    (*=== VARIABLE LIST ===============================================================================*)
    zz_VariableList :   ARRAY[1..zz_VARIABLECOUNT] OF MBCFG_typVARIABLE :=
    (    DataType        := MBCFG_TYPE_REAL,
        ByteOrder       := MBCFG_BYTE_ORDER_3,
        BitSize         := 32,
        ptVar           := 0,
        ReadJobIndex    := 1,
        ReadStartBitNo  := 256,
        WriteJobIndex   := 0,
        WriteStartBitNo := 0 ),
    (    DataType        := MBCFG_TYPE_REAL,
        ByteOrder       := MBCFG_BYTE_ORDER_3,
        BitSize         := 32,
        ptVar           := 0,
        ReadJobIndex    := 1,
        ReadStartBitNo  := 288,
        WriteJobIndex   := 0,
        WriteStartBitNo := 0 ),
    (    DataType        := MBCFG_TYPE_REAL,
        ByteOrder       := MBCFG_BYTE_ORDER_3,
        BitSize         := 32,
        ptVar           := 0,
        ReadJobIndex    := 1,
        ReadStartBitNo  := 320,
        WriteJobIndex   := 0,
        WriteStartBitNo := 0 ),
    (    DataType        := MBCFG_TYPE_REAL,
        ByteOrder       := MBCFG_BYTE_ORDER_3,
        BitSize         := 32,
        ptVar           := 0,
        ReadJobIndex    := 1,
        ReadStartBitNo  := 384,
        WriteJobIndex   := 0,
        WriteStartBitNo := 0 ),
    (    DataType        := MBCFG_TYPE_REAL,
        ByteOrder       := MBCFG_BYTE_ORDER_3,
        BitSize         := 32,
        ptVar           := 0,
        ReadJobIndex    := 1,
        ReadStartBitNo  := 416,
        WriteJobIndex   := 0,
        WriteStartBitNo := 0 ),
    (    DataType        := MBCFG_TYPE_REAL,
        ByteOrder       := MBCFG_BYTE_ORDER_3,
        BitSize         := 32,
        ptVar           := 0,
        ReadJobIndex    := 1,
        ReadStartBitNo  := 448,
        WriteJobIndex   := 0,
        WriteStartBitNo := 0 ),
    (    DataType        := MBCFG_TYPE_REAL,
        ByteOrder       := MBCFG_BYTE_ORDER_3,
        BitSize         := 32,
        ptVar           := 0,
        ReadJobIndex    := 1,
        ReadStartBitNo  := 0,
        WriteJobIndex   := 0,
        WriteStartBitNo := 0 ),
    (    DataType        := MBCFG_TYPE_REAL,
        ByteOrder       := MBCFG_BYTE_ORDER_3,
        BitSize         := 32,
        ptVar           := 0,
        ReadJobIndex    := 1,
        ReadStartBitNo  := 32,
        WriteJobIndex   := 0,
        WriteStartBitNo := 0 ),
    (    DataType        := MBCFG_TYPE_REAL,
        ByteOrder       := MBCFG_BYTE_ORDER_3,
        BitSize         := 32,
        ptVar           := 0,
        ReadJobIndex    := 1,
        ReadStartBitNo  := 64,
        WriteJobIndex   := 0,
        WriteStartBitNo := 0 ),
    (    DataType        := MBCFG_TYPE_REAL,
        ByteOrder       := MBCFG_BYTE_ORDER_3,
        BitSize         := 32,
        ptVar           := 0,
        ReadJobIndex    := 1,
        ReadStartBitNo  := 96,
        WriteJobIndex   := 0,
        WriteStartBitNo := 0 ),
    (    DataType        := MBCFG_TYPE_REAL,
        ByteOrder       := MBCFG_BYTE_ORDER_3,
        BitSize         := 32,
        ptVar           := 0,
        ReadJobIndex    := 1,
        ReadStartBitNo  := 128,
        WriteJobIndex   := 0,
        WriteStartBitNo := 0 ),
    (    DataType        := MBCFG_TYPE_REAL,
        ByteOrder       := MBCFG_BYTE_ORDER_3,
        BitSize         := 32,
        ptVar           := 0,
        ReadJobIndex    := 1,
        ReadStartBitNo  := 160,
        WriteJobIndex   := 0,
        WriteStartBitNo := 0 ),
    (    DataType        := MBCFG_TYPE_REAL,
        ByteOrder       := MBCFG_BYTE_ORDER_3,
        BitSize         := 32,
        ptVar           := 0,
        ReadJobIndex    := 1,
        ReadStartBitNo  := 192,
        WriteJobIndex   := 0,
        WriteStartBitNo := 0 ),
    (    DataType        := MBCFG_TYPE_REAL,
        ByteOrder       := MBCFG_BYTE_ORDER_3,
        BitSize         := 32,
        ptVar           := 0,
        ReadJobIndex    := 1,
        ReadStartBitNo  := 224,
        WriteJobIndex   := 0,
        WriteStartBitNo := 0 ),
    (    DataType        := MBCFG_TYPE_REAL,
        ByteOrder       := MBCFG_BYTE_ORDER_3,
        BitSize         := 32,
        ptVar           := 0,
        ReadJobIndex    := 2,
        ReadStartBitNo  := 416,
        WriteJobIndex   := 0,
        WriteStartBitNo := 0 ),
    (    DataType        := MBCFG_TYPE_REAL,
        ByteOrder       := MBCFG_BYTE_ORDER_3,
        BitSize         := 32,
        ptVar           := 0,
        ReadJobIndex    := 2,
        ReadStartBitNo  := 0,
        WriteJobIndex   := 0,
        WriteStartBitNo := 0 ),
    (    DataType        := MBCFG_TYPE_REAL,
        ByteOrder       := MBCFG_BYTE_ORDER_3,
        BitSize         := 32,
        ptVar           := 0,
        ReadJobIndex    := 2,
        ReadStartBitNo  := 32,
        WriteJobIndex   := 0,
        WriteStartBitNo := 0 ),
    (    DataType        := MBCFG_TYPE_REAL,
        ByteOrder       := MBCFG_BYTE_ORDER_3,
        BitSize         := 32,
        ptVar           := 0,
        ReadJobIndex    := 2,
        ReadStartBitNo  := 64,
        WriteJobIndex   := 0,
        WriteStartBitNo := 0 ),
    (    DataType        := MBCFG_TYPE_REAL,
        ByteOrder       := MBCFG_BYTE_ORDER_3,
        BitSize         := 32,
        ptVar           := 0,
        ReadJobIndex    := 2,
        ReadStartBitNo  := 256,
        WriteJobIndex   := 0,
        WriteStartBitNo := 0 ),
    (    DataType        := MBCFG_TYPE_REAL,
        ByteOrder       := MBCFG_BYTE_ORDER_3,
        BitSize         := 32,
        ptVar           := 0,
        ReadJobIndex    := 3,
        ReadStartBitNo  := 0,
        WriteJobIndex   := 0,
        WriteStartBitNo := 0 ),
    (    DataType        := MBCFG_TYPE_REAL,
        ByteOrder       := MBCFG_BYTE_ORDER_3,
        BitSize         := 32,
        ptVar           := 0,
        ReadJobIndex    := 3,
        ReadStartBitNo  := 128,
        WriteJobIndex   := 0,
        WriteStartBitNo := 0 )

                        ;
    (*=================================================================================================*)

    (*=== JOB LIST ====================================================================================*)
    zz_JobList     :   ARRAY[1..zz_JOBCOUNT] OF MBCFG_typCOM_JOB :=
     (   Functioncode            := 3,
        ReadStartAddress        := 2053,
        ReadQuantity            := 30,
        WriteStartAddress       := 0,
        WriteQuantity           := 0,
        ptReadData              := 0, 
        ptWriteData             := 0 ),
     (   Functioncode            := 3,
        ReadStartAddress        := 2159,
        ReadQuantity            := 28,
        WriteStartAddress       := 0,
        WriteQuantity           := 0,
        ptReadData              := 0, 
        ptWriteData             := 0 ),
     (   Functioncode            := 3,
        ReadStartAddress        := 2105,
        ReadQuantity            := 10,
        WriteStartAddress       := 0,
        WriteQuantity           := 0,
        ptReadData              := 0, 
        ptWriteData             := 0 )

                        ;
    (*=================================================================================================*)

    (*=== DATA FIELDS =================================================================================*)
     zz_DataField_1_Read       :       ARRAY[1..30] OF WORD;
     zz_DataField_2_Read       :       ARRAY[1..28] OF WORD;
     zz_DataField_3_Read       :       ARRAY[1..10] OF WORD;
	
    (*=================================================================================================*)

    (*=== MODBUS MASTER =====================================*)
    zz_MBCFG_MASTER_ETH :       MBCFG_MASTER_UDP;
    (*=======================================================*)

END_VAR
(*--- for each variable -------------------------*)
   zz_VariableList[1].ptVar := ADR(PactiveL1);
   zz_VariableList[2].ptVar := ADR(PactiveL2);
   zz_VariableList[3].ptVar := ADR(PactiveL3);
   zz_VariableList[4].ptVar := ADR(PreactiveL1);
   zz_VariableList[5].ptVar := ADR(PreactiveL2);
   zz_VariableList[6].ptVar := ADR(PreactiveL3);
   zz_VariableList[7].ptVar := ADR(VoltageL1);
   zz_VariableList[8].ptVar := ADR(VoltageL2);
   zz_VariableList[9].ptVar := ADR(VoltageL3);
   zz_VariableList[10].ptVar := ADR(VoltageL4);
   zz_VariableList[11].ptVar := ADR(PhaseCurrentL1);
   zz_VariableList[12].ptVar := ADR(PhaseCurrentL2);
   zz_VariableList[13].ptVar := ADR(PhaseCurrentL3);
   zz_VariableList[14].ptVar := ADR(PhaseCurrentLN);
   zz_VariableList[15].ptVar := ADR(FieldRotation);
   zz_VariableList[16].ptVar := ADR(CosPihL1);
   zz_VariableList[17].ptVar := ADR(CosPihL2);
   zz_VariableList[18].ptVar := ADR(CosPihL3);
   zz_VariableList[19].ptVar := ADR(Frequency);
   zz_VariableList[20].ptVar := ADR(PactivetTot);
   zz_VariableList[21].ptVar := ADR(PactivetTotL4);

(*-----------------------------------------------*)

(*--- for each job -----------------------------------*)
zz_JobList[1].ptReadData   := ADR(zz_DataField_1_Read);
zz_JobList[2].ptReadData   := ADR(zz_DataField_2_Read);
zz_JobList[3].ptReadData   := ADR(zz_DataField_3_Read);

(*----------------------------------------------------*)


(*#### START OF FIXED CODE #####################################*)
zz_MBCFG_MASTER_ETH(	strIpAddress    := MBCFG_IpAddress,                 (* fixed entry     *)
                        uiPort          := MBCFG_Port,                      (* fixed entry     *)
                        bUnitID         := MBCFG_UnitID,                    (* fixed entry     *)
                        tTimeOut        := MBCFG_TimeOut,                   (* fixed entry     *)
                        iVariableCount  := zz_VARIABLECOUNT,
                        ptVariableList  := ADR(zz_VariableList),
                        iJobCount       := zz_JOBCOUNT,
                        ptJobList       := ADR(zz_JobList),
                        tRequestDelay   := MBCFG_RequestDelay,              (* fixed entry     *)
                        eError          => MBCFG_Error,                     (* fixed entry     *)
                        LastJob         => MBCFG_LastJob                    (* fixed entry     *)
                    );
(*##############################################################*)
END_PROGRAM

(* POU 01. PowerQualityMeasurements/PQ_1, FBD *)
PROGRAM PQ_1
VAR
	abProcessImageInput	AT %IW12			: ARRAY[0..23] OF BYTE;
	abProcessImageOutput 	AT %QW20		: ARRAY[0..23] OF BYTE;

	bToken										: BYTE;

	State_750_495 							: Fb_750_495_State;
		typ_750_495_State 						: typ_750_495_State;

	Configuration_750_495					: Fb_750_495_Configuration;
		typConfig_750_495						: typConfig_750_495;
		xReadyConfig								: BOOL;
		bFeedbackConfig							: BYTE;

	AC_Compact_01_750_495				: Fb_750_495_AC_Compact_01;
		rTotalActivePower							: REAL;
		rTotalReactivePower						: REAL;
		rTotalApparentPower						: REAL;
		rTotalPowerFactorPF						: REAL;
		rTotalActiveEnergy							: REAL;
		rTotalReactiveEnergy						: REAL;
		rTotalApparentEnergy						: REAL;
		rCurrentN									: REAL;
		xRotatingField								: BOOL;
		arCurrent									: ARRAY[1..3] OF REAL;
		axOvercurrent								: ARRAY[1..3] OF BOOL;
		arVoltage_L_N							: ARRAY[1..3] OF REAL;
		axUndervoltage							: ARRAY[1..3] OF BOOL;
		axOvervoltage								: ARRAY[1..3] OF BOOL;
		arActivePower								: ARRAY[1..3] OF REAL;
		arReactivePower							: ARRAY[1..3] OF REAL;
		arApparentPower							: ARRAY[1..3] OF REAL;
		arCosPhi									: ARRAY[1..3] OF REAL;
		arPowerFactorPF							: ARRAY[1..3] OF REAL;
		arFrequency								: ARRAY[1..3] OF REAL;
		axNoZero									: ARRAY[1..3] OF BOOL;
		axVoltSag									: ARRAY[1..3] OF BOOL;
		ai4Quadrant								: ARRAY[1..3] OF INT;

		xReadyCompact_01						: BOOL;
		abFeedbackCompact_01					: ARRAY[1..8] OF BYTE;


END_VAR
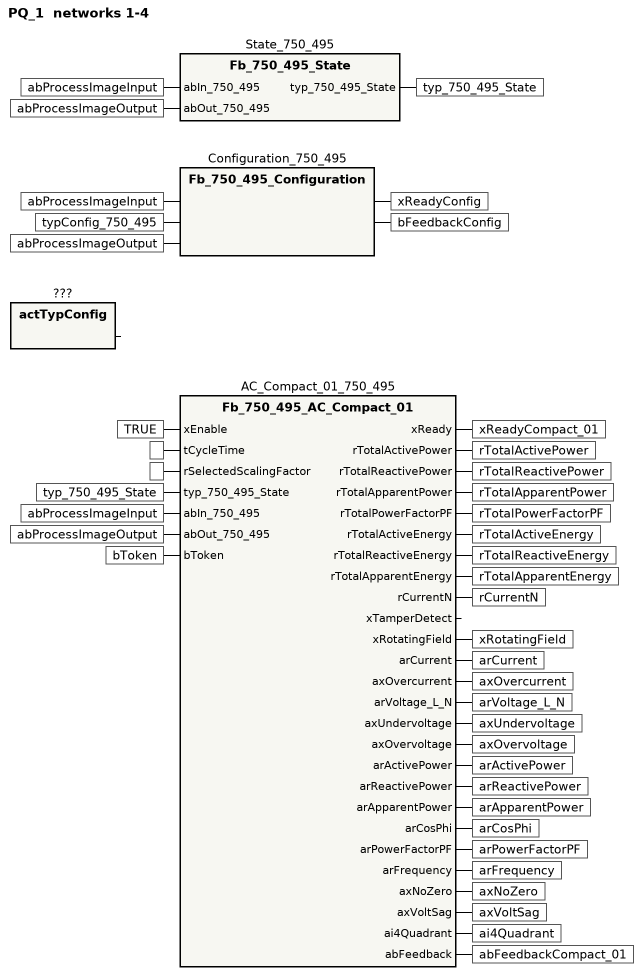
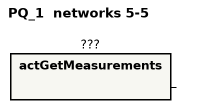
_FBD_ (* Function Block Diagram *)
NETWORK 1
	State_750_495:Fb_750_495_State(abIn_750_495: abProcessImageInput, abOut_750_495: abProcessImageOutput) => typ_750_495_State
NETWORK 2
	Configuration_750_495:Fb_750_495_Configuration(abProcessImageInput, typConfig_750_495, abProcessImageOutput, out 2 => bFeedbackConfig) => xReadyConfig
NETWORK 3
	???:actTypConfig()
NETWORK 4
	AC_Compact_01_750_495:Fb_750_495_AC_Compact_01(xEnable: TRUE, tCycleTime: , rSelectedScalingFactor: , typ_750_495_State: typ_750_495_State, abIn_750_495: abProcessImageInput, abOut_750_495: abProcessImageOutput, bToken: bToken, rTotalActivePower => rTotalActivePower, rTotalReactivePower => rTotalReactivePower, rTotalApparentPower => rTotalApparentPower, rTotalPowerFactorPF => rTotalPowerFactorPF, rTotalActiveEnergy => rTotalActiveEnergy, rTotalReactiveEnergy => rTotalReactiveEnergy, rTotalApparentEnergy => rTotalApparentEnergy, rCurrentN => rCurrentN, xRotatingField => xRotatingField, arCurrent => arCurrent, axOvercurrent => axOvercurrent, arVoltage_L_N => arVoltage_L_N, axUndervoltage => axUndervoltage, axOvervoltage => axOvervoltage, arActivePower => arActivePower, arReactivePower => arReactivePower, arApparentPower => arApparentPower, arCosPhi => arCosPhi, arPowerFactorPF => arPowerFactorPF, arFrequency => arFrequency, axNoZero => axNoZero, axVoltSag => axVoltSag, ai4Quadrant => ai4Quadrant, abFeedback => abFeedbackCompact_01) => xReadyCompact_01
NETWORK 5
	???:actGetMeasurements()
_END_FBD_
(* the same logic as Structured Text *)
(* Network 1 *)
State_750_495(abIn_750_495 := abProcessImageInput, abOut_750_495 := abProcessImageOutput);
typ_750_495_State := State_750_495.typ_750_495_State;
(* Network 2: see the listing above *)
(* Network 3: see the listing above *)
(* Network 4: see the listing above *)
(* Network 5: see the listing above *)
END_PROGRAM
ACTION actGetMeasurements:
arMeasurementsGroup1[1] := arActivePower[1];
arMeasurementsGroup1[2] := arActivePower[2];
arMeasurementsGroup1[3] := arActivePower[3];
arMeasurementsGroup1[4] := arReactivePower[1];
arMeasurementsGroup1[5] := arReactivePower[2];
arMeasurementsGroup1[6] := arReactivePower[3];
arMeasurementsGroup1[7] := arVoltage_L_N[1];
arMeasurementsGroup1[8] := arVoltage_L_N[2];
arMeasurementsGroup1[9] := arVoltage_L_N[3];
arMeasurementsGroup1[10] := arCurrent[1];
arMeasurementsGroup1[11] := arCurrent[2];
arMeasurementsGroup1[12] := arCurrent[3];
arMeasurementsGroup1[13] := arFrequency[1];
arMeasurementsGroup1[14] := arFrequency[2];
arMeasurementsGroup1[15] := arFrequency[3];
arMeasurementsGroup1[16] := rTotalActiveEnergy;
arMeasurementsGroup1[17] := BOOL_TO_REAL(xRotatingField);
arMeasurementsGroup1[18] := rTotalReactiveEnergy;
END_ACTION
ACTION actTypConfig:
typConfig_750_495.typChannelConfig[1].xEnableUserScaling:= TRUE;
typConfig_750_495.typChannelConfig[1].wCurrentTransformerRatio :=CurrentRatioPQ1;

typConfig_750_495.typChannelConfig[2].xEnableUserScaling:= TRUE;
typConfig_750_495.typChannelConfig[2].wCurrentTransformerRatio :=CurrentRatioPQ1;

typConfig_750_495.typChannelConfig[3].xEnableUserScaling:= TRUE;
typConfig_750_495.typChannelConfig[3].wCurrentTransformerRatio :=CurrentRatioPQ1;

typConfig_750_495.xWriteConfig := TRUE;
END_ACTION

(* POU 01. PowerQualityMeasurements/PQ_2, FBD *)
PROGRAM PQ_2
VAR
	abProcessImageInput	AT %IW24			: ARRAY[0..23] OF BYTE;
	abProcessImageOutput 	AT %QW32 			: ARRAY[0..23] OF BYTE;

	bToken										: BYTE;

	State_750_495 							: Fb_750_495_State;
		typ_750_495_State 						: typ_750_495_State;

	Configuration_750_495					: Fb_750_495_Configuration;
		typConfig_750_495						: typConfig_750_495;
		xReadyConfig								: BOOL;
		bFeedbackConfig							: BYTE;

	AC_Compact_01_750_495				: Fb_750_495_AC_Compact_01;
		rTotalActivePower							: REAL;
		rTotalReactivePower						: REAL;
		rTotalApparentPower						: REAL;
		rTotalPowerFactorPF						: REAL;
		rTotalActiveEnergy							: REAL;
		rTotalReactiveEnergy						: REAL;
		rTotalApparentEnergy						: REAL;
		rCurrentN									: REAL;
		xRotatingField								: BOOL;
		arCurrent									: ARRAY[1..3] OF REAL;
		axOvercurrent								: ARRAY[1..3] OF BOOL;
		arVoltage_L_N							: ARRAY[1..3] OF REAL;
		axUndervoltage							: ARRAY[1..3] OF BOOL;
		axOvervoltage								: ARRAY[1..3] OF BOOL;
		arActivePower								: ARRAY[1..3] OF REAL;
		arReactivePower							: ARRAY[1..3] OF REAL;
		arApparentPower							: ARRAY[1..3] OF REAL;
		arCosPhi									: ARRAY[1..3] OF REAL;
		arPowerFactorPF							: ARRAY[1..3] OF REAL;
		arFrequency								: ARRAY[1..3] OF REAL;
		axNoZero									: ARRAY[1..3] OF BOOL;
		axVoltSag									: ARRAY[1..3] OF BOOL;
		ai4Quadrant								: ARRAY[1..3] OF INT;

		xReadyCompact_01						: BOOL;
		abFeedbackCompact_01					: ARRAY[1..8] OF BYTE;


END_VAR
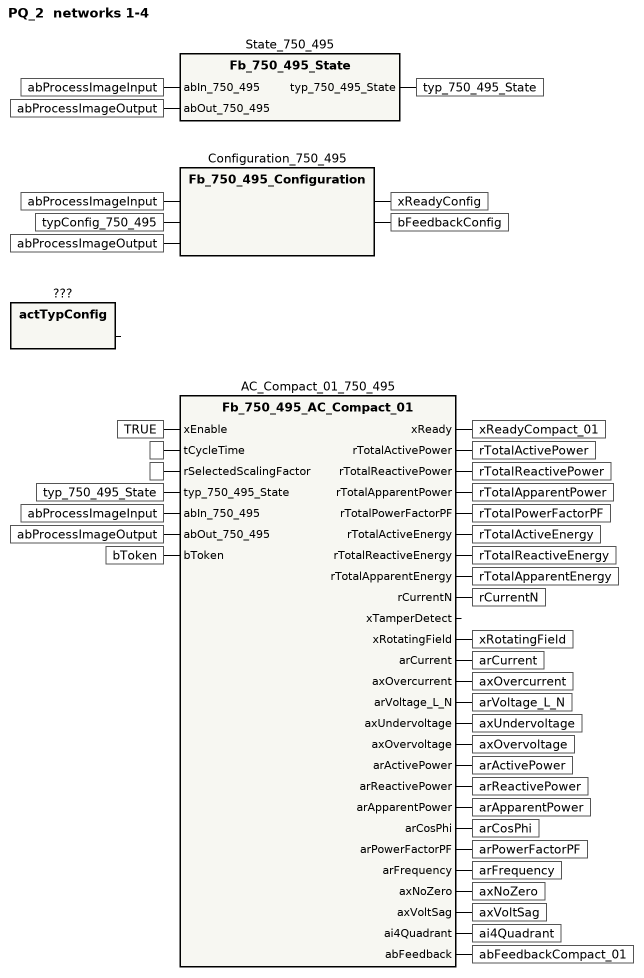
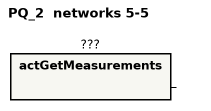
_FBD_ (* Function Block Diagram *)
NETWORK 1
	State_750_495:Fb_750_495_State(abIn_750_495: abProcessImageInput, abOut_750_495: abProcessImageOutput) => typ_750_495_State
NETWORK 2
	Configuration_750_495:Fb_750_495_Configuration(abProcessImageInput, typConfig_750_495, abProcessImageOutput, out 2 => bFeedbackConfig) => xReadyConfig
NETWORK 3
	???:actTypConfig()
NETWORK 4
	AC_Compact_01_750_495:Fb_750_495_AC_Compact_01(xEnable: TRUE, tCycleTime: , rSelectedScalingFactor: , typ_750_495_State: typ_750_495_State, abIn_750_495: abProcessImageInput, abOut_750_495: abProcessImageOutput, bToken: bToken, rTotalActivePower => rTotalActivePower, rTotalReactivePower => rTotalReactivePower, rTotalApparentPower => rTotalApparentPower, rTotalPowerFactorPF => rTotalPowerFactorPF, rTotalActiveEnergy => rTotalActiveEnergy, rTotalReactiveEnergy => rTotalReactiveEnergy, rTotalApparentEnergy => rTotalApparentEnergy, rCurrentN => rCurrentN, xRotatingField => xRotatingField, arCurrent => arCurrent, axOvercurrent => axOvercurrent, arVoltage_L_N => arVoltage_L_N, axUndervoltage => axUndervoltage, axOvervoltage => axOvervoltage, arActivePower => arActivePower, arReactivePower => arReactivePower, arApparentPower => arApparentPower, arCosPhi => arCosPhi, arPowerFactorPF => arPowerFactorPF, arFrequency => arFrequency, axNoZero => axNoZero, axVoltSag => axVoltSag, ai4Quadrant => ai4Quadrant, abFeedback => abFeedbackCompact_01) => xReadyCompact_01
NETWORK 5
	???:actGetMeasurements()
_END_FBD_
(* the same logic as Structured Text *)
(* Network 1 *)
State_750_495(abIn_750_495 := abProcessImageInput, abOut_750_495 := abProcessImageOutput);
typ_750_495_State := State_750_495.typ_750_495_State;
(* Network 2: see the listing above *)
(* Network 3: see the listing above *)
(* Network 4: see the listing above *)
(* Network 5: see the listing above *)
END_PROGRAM
ACTION actGetMeasurements:
arMeasurementsGroup2[1] := arActivePower[1];
arMeasurementsGroup2[2] := arActivePower[2];
arMeasurementsGroup2[3] := arActivePower[3];
arMeasurementsGroup2[4] := arReactivePower[1];
arMeasurementsGroup2[5] := arReactivePower[2];
arMeasurementsGroup2[6] := arReactivePower[3];
arMeasurementsGroup2[7] := arVoltage_L_N[1];
arMeasurementsGroup2[8] := arVoltage_L_N[2];
arMeasurementsGroup2[9] := arVoltage_L_N[3];
arMeasurementsGroup2[10] := arCurrent[1];
arMeasurementsGroup2[11] := arCurrent[2];
arMeasurementsGroup2[12] := arCurrent[3];
arMeasurementsGroup2[13] := arFrequency[1];
arMeasurementsGroup2[14] := arFrequency[2];
arMeasurementsGroup2[15] := arFrequency[3];
arMeasurementsGroup2[16] := rTotalActiveEnergy;
arMeasurementsGroup2[17] := BOOL_TO_REAL(xRotatingField);
arMeasurementsGroup2[18] := rTotalReactiveEnergy;
END_ACTION
ACTION actTypConfig:
typConfig_750_495.typChannelConfig[1].xEnableUserScaling:= TRUE;
typConfig_750_495.typChannelConfig[1].wCurrentTransformerRatio :=CurrentRatioPQ2;

typConfig_750_495.typChannelConfig[2].xEnableUserScaling:= TRUE;
typConfig_750_495.typChannelConfig[2].wCurrentTransformerRatio :=CurrentRatioPQ2;

typConfig_750_495.typChannelConfig[3].xEnableUserScaling:= TRUE;
typConfig_750_495.typChannelConfig[3].wCurrentTransformerRatio :=CurrentRatioPQ2;

typConfig_750_495.xWriteConfig := TRUE;
END_ACTION

(* POU 01. PowerQualityMeasurements/PQ_3, FBD *)
PROGRAM PQ_3
VAR
	abProcessImageInput	AT %IW36			: ARRAY[0..23] OF BYTE;
	abProcessImageOutput 	AT %QW44		: ARRAY[0..23] OF BYTE;

	bToken										: BYTE;

	State_750_495 							: Fb_750_495_State;
		typ_750_495_State 						: typ_750_495_State;

	Configuration_750_495					: Fb_750_495_Configuration;
		typConfig_750_495						: typConfig_750_495;
		xReadyConfig								: BOOL;
		bFeedbackConfig							: BYTE;

	AC_Compact_01_750_495				: Fb_750_495_AC_Compact_01;
		rTotalActivePower							: REAL;
		rTotalReactivePower						: REAL;
		rTotalApparentPower						: REAL;
		rTotalPowerFactorPF						: REAL;
		rTotalActiveEnergy							: REAL;
		rTotalReactiveEnergy						: REAL;
		rTotalApparentEnergy						: REAL;
		rCurrentN									: REAL;
		xRotatingField								: BOOL;
		arCurrent									: ARRAY[1..3] OF REAL;
		axOvercurrent								: ARRAY[1..3] OF BOOL;
		arVoltage_L_N							: ARRAY[1..3] OF REAL;
		axUndervoltage							: ARRAY[1..3] OF BOOL;
		axOvervoltage								: ARRAY[1..3] OF BOOL;
		arActivePower								: ARRAY[1..3] OF REAL;
		arReactivePower							: ARRAY[1..3] OF REAL;
		arApparentPower							: ARRAY[1..3] OF REAL;
		arCosPhi									: ARRAY[1..3] OF REAL;
		arPowerFactorPF							: ARRAY[1..3] OF REAL;
		arFrequency								: ARRAY[1..3] OF REAL;
		axNoZero									: ARRAY[1..3] OF BOOL;
		axVoltSag									: ARRAY[1..3] OF BOOL;
		ai4Quadrant								: ARRAY[1..3] OF INT;

		xReadyCompact_01						: BOOL;
		abFeedbackCompact_01					: ARRAY[1..8] OF BYTE;


END_VAR
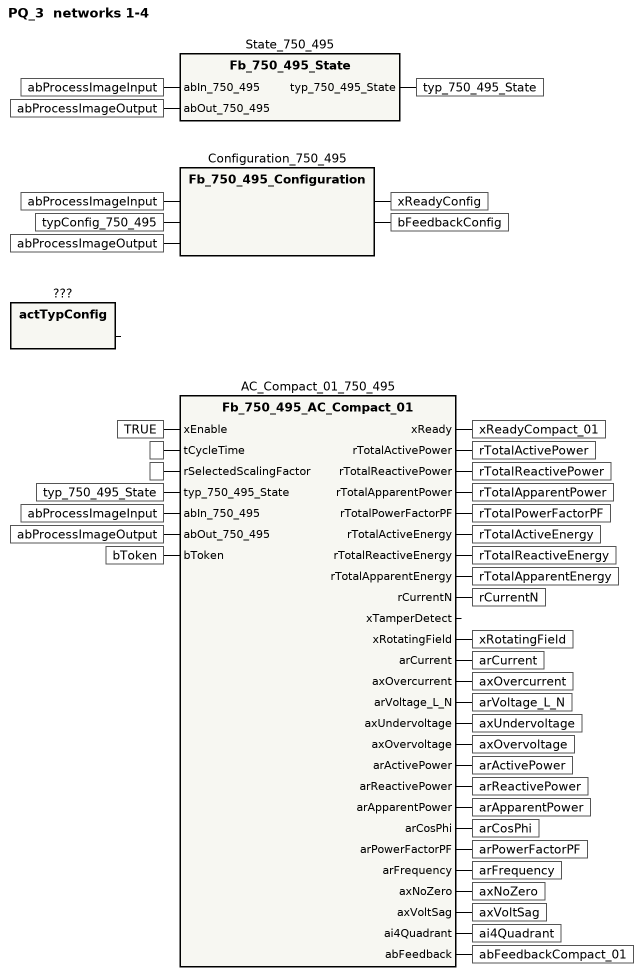
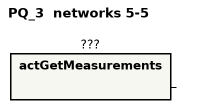
_FBD_ (* Function Block Diagram *)
NETWORK 1
	State_750_495:Fb_750_495_State(abIn_750_495: abProcessImageInput, abOut_750_495: abProcessImageOutput) => typ_750_495_State
NETWORK 2
	Configuration_750_495:Fb_750_495_Configuration(abProcessImageInput, typConfig_750_495, abProcessImageOutput, out 2 => bFeedbackConfig) => xReadyConfig
NETWORK 3
	???:actTypConfig()
NETWORK 4
	AC_Compact_01_750_495:Fb_750_495_AC_Compact_01(xEnable: TRUE, tCycleTime: , rSelectedScalingFactor: , typ_750_495_State: typ_750_495_State, abIn_750_495: abProcessImageInput, abOut_750_495: abProcessImageOutput, bToken: bToken, rTotalActivePower => rTotalActivePower, rTotalReactivePower => rTotalReactivePower, rTotalApparentPower => rTotalApparentPower, rTotalPowerFactorPF => rTotalPowerFactorPF, rTotalActiveEnergy => rTotalActiveEnergy, rTotalReactiveEnergy => rTotalReactiveEnergy, rTotalApparentEnergy => rTotalApparentEnergy, rCurrentN => rCurrentN, xRotatingField => xRotatingField, arCurrent => arCurrent, axOvercurrent => axOvercurrent, arVoltage_L_N => arVoltage_L_N, axUndervoltage => axUndervoltage, axOvervoltage => axOvervoltage, arActivePower => arActivePower, arReactivePower => arReactivePower, arApparentPower => arApparentPower, arCosPhi => arCosPhi, arPowerFactorPF => arPowerFactorPF, arFrequency => arFrequency, axNoZero => axNoZero, axVoltSag => axVoltSag, ai4Quadrant => ai4Quadrant, abFeedback => abFeedbackCompact_01) => xReadyCompact_01
NETWORK 5
	???:actGetMeasurements()
_END_FBD_
(* the same logic as Structured Text *)
(* Network 1 *)
State_750_495(abIn_750_495 := abProcessImageInput, abOut_750_495 := abProcessImageOutput);
typ_750_495_State := State_750_495.typ_750_495_State;
(* Network 2: see the listing above *)
(* Network 3: see the listing above *)
(* Network 4: see the listing above *)
(* Network 5: see the listing above *)
END_PROGRAM
ACTION actGetMeasurements:
arMeasurementsGroup3[1] := arActivePower[1];
arMeasurementsGroup3[2] := arActivePower[2];
arMeasurementsGroup3[3] := arActivePower[3];
arMeasurementsGroup3[4] := arReactivePower[1];
arMeasurementsGroup3[5] := arReactivePower[2];
arMeasurementsGroup3[6] := arReactivePower[3];
arMeasurementsGroup3[7] := arVoltage_L_N[1];
arMeasurementsGroup3[8] := arVoltage_L_N[2];
arMeasurementsGroup3[9] := arVoltage_L_N[3];
arMeasurementsGroup3[10] := arCurrent[1];
arMeasurementsGroup3[11] := arCurrent[2];
arMeasurementsGroup3[12] := arCurrent[3];
arMeasurementsGroup3[13] := arFrequency[1];
arMeasurementsGroup3[14] := arFrequency[2];
arMeasurementsGroup3[15] := arFrequency[3];
arMeasurementsGroup3[16] := rTotalActiveEnergy;
arMeasurementsGroup3[17] := BOOL_TO_REAL(xRotatingField);
arMeasurementsGroup3[18] := rTotalReactiveEnergy;
END_ACTION
ACTION actTypConfig:
typConfig_750_495.typChannelConfig[1].xEnableUserScaling:= TRUE;
typConfig_750_495.typChannelConfig[1].wCurrentTransformerRatio :=CurrentRatioPQ3;

typConfig_750_495.typChannelConfig[2].xEnableUserScaling:= TRUE;
typConfig_750_495.typChannelConfig[2].wCurrentTransformerRatio :=CurrentRatioPQ3;

typConfig_750_495.typChannelConfig[3].xEnableUserScaling:= TRUE;
typConfig_750_495.typChannelConfig[3].wCurrentTransformerRatio :=CurrentRatioPQ3;

typConfig_750_495.xWriteConfig := TRUE;
END_ACTION

(* POU 01. PowerQualityMeasurements/PQ_4, FBD *)
PROGRAM PQ_4
VAR
	abProcessImageInput	AT %IW48			: ARRAY[0..23] OF BYTE;
	abProcessImageOutput 	AT %QW56		: ARRAY[0..23] OF BYTE;

	bToken										: BYTE;

	State_750_495 							: Fb_750_495_State;
		typ_750_495_State 						: typ_750_495_State;

	Configuration_750_495					: Fb_750_495_Configuration;
		typConfig_750_495						: typConfig_750_495;
		xReadyConfig								: BOOL;
		bFeedbackConfig							: BYTE;

	AC_Compact_01_750_495				: Fb_750_495_AC_Compact_01;
		rTotalActivePower							: REAL;
		rTotalReactivePower						: REAL;
		rTotalApparentPower						: REAL;
		rTotalPowerFactorPF						: REAL;
		rTotalActiveEnergy							: REAL;
		rTotalReactiveEnergy						: REAL;
		rTotalApparentEnergy						: REAL;
		rCurrentN									: REAL;
		xRotatingField								: BOOL;
		arCurrent									: ARRAY[1..3] OF REAL;
		axOvercurrent								: ARRAY[1..3] OF BOOL;
		arVoltage_L_N							: ARRAY[1..3] OF REAL;
		axUndervoltage							: ARRAY[1..3] OF BOOL;
		axOvervoltage								: ARRAY[1..3] OF BOOL;
		arActivePower								: ARRAY[1..3] OF REAL;
		arReactivePower							: ARRAY[1..3] OF REAL;
		arApparentPower							: ARRAY[1..3] OF REAL;
		arCosPhi									: ARRAY[1..3] OF REAL;
		arPowerFactorPF							: ARRAY[1..3] OF REAL;
		arFrequency								: ARRAY[1..3] OF REAL;
		axNoZero									: ARRAY[1..3] OF BOOL;
		axVoltSag									: ARRAY[1..3] OF BOOL;
		ai4Quadrant								: ARRAY[1..3] OF INT;

		xReadyCompact_01						: BOOL;
		abFeedbackCompact_01					: ARRAY[1..8] OF BYTE;


END_VAR
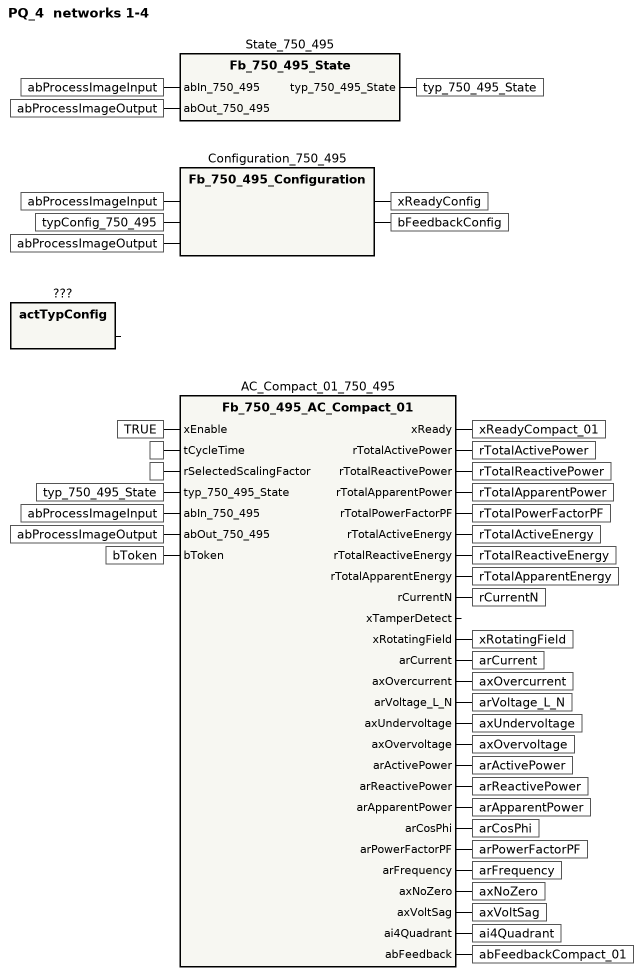
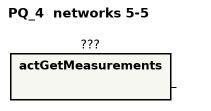
_FBD_ (* Function Block Diagram *)
NETWORK 1
	State_750_495:Fb_750_495_State(abIn_750_495: abProcessImageInput, abOut_750_495: abProcessImageOutput) => typ_750_495_State
NETWORK 2
	Configuration_750_495:Fb_750_495_Configuration(abProcessImageInput, typConfig_750_495, abProcessImageOutput, out 2 => bFeedbackConfig) => xReadyConfig
NETWORK 3
	???:actTypConfig()
NETWORK 4
	AC_Compact_01_750_495:Fb_750_495_AC_Compact_01(xEnable: TRUE, tCycleTime: , rSelectedScalingFactor: , typ_750_495_State: typ_750_495_State, abIn_750_495: abProcessImageInput, abOut_750_495: abProcessImageOutput, bToken: bToken, rTotalActivePower => rTotalActivePower, rTotalReactivePower => rTotalReactivePower, rTotalApparentPower => rTotalApparentPower, rTotalPowerFactorPF => rTotalPowerFactorPF, rTotalActiveEnergy => rTotalActiveEnergy, rTotalReactiveEnergy => rTotalReactiveEnergy, rTotalApparentEnergy => rTotalApparentEnergy, rCurrentN => rCurrentN, xRotatingField => xRotatingField, arCurrent => arCurrent, axOvercurrent => axOvercurrent, arVoltage_L_N => arVoltage_L_N, axUndervoltage => axUndervoltage, axOvervoltage => axOvervoltage, arActivePower => arActivePower, arReactivePower => arReactivePower, arApparentPower => arApparentPower, arCosPhi => arCosPhi, arPowerFactorPF => arPowerFactorPF, arFrequency => arFrequency, axNoZero => axNoZero, axVoltSag => axVoltSag, ai4Quadrant => ai4Quadrant, abFeedback => abFeedbackCompact_01) => xReadyCompact_01
NETWORK 5
	???:actGetMeasurements()
_END_FBD_
(* the same logic as Structured Text *)
(* Network 1 *)
State_750_495(abIn_750_495 := abProcessImageInput, abOut_750_495 := abProcessImageOutput);
typ_750_495_State := State_750_495.typ_750_495_State;
(* Network 2: see the listing above *)
(* Network 3: see the listing above *)
(* Network 4: see the listing above *)
(* Network 5: see the listing above *)
END_PROGRAM
ACTION actGetMeasurements:
arMeasurementsGroup4[1] := arActivePower[1];
arMeasurementsGroup4[2] := arActivePower[2];
arMeasurementsGroup4[3] := arActivePower[3];
arMeasurementsGroup4[4] := arReactivePower[1];
arMeasurementsGroup4[5] := arReactivePower[2];
arMeasurementsGroup4[6] := arReactivePower[3];
arMeasurementsGroup4[7] := arVoltage_L_N[1];
arMeasurementsGroup4[8] := arVoltage_L_N[2];
arMeasurementsGroup4[9] := arVoltage_L_N[3];
arMeasurementsGroup4[10] := arCurrent[1];
arMeasurementsGroup4[11] := arCurrent[2];
arMeasurementsGroup4[12] := arCurrent[3];
arMeasurementsGroup4[13] := arFrequency[1];
arMeasurementsGroup4[14] := arFrequency[2];
arMeasurementsGroup4[15] := arFrequency[3];
arMeasurementsGroup4[16] := rTotalActiveEnergy;
arMeasurementsGroup4[17] := BOOL_TO_REAL(xRotatingField);
arMeasurementsGroup4[18] := rTotalReactiveEnergy;
END_ACTION
ACTION actTypConfig:
typConfig_750_495.typChannelConfig[1].xEnableUserScaling:= TRUE;
typConfig_750_495.typChannelConfig[1].wCurrentTransformerRatio :=CurrentRatioPQ4;

typConfig_750_495.typChannelConfig[2].xEnableUserScaling:= TRUE;
typConfig_750_495.typChannelConfig[2].wCurrentTransformerRatio :=CurrentRatioPQ4;

typConfig_750_495.typChannelConfig[3].xEnableUserScaling:= TRUE;
typConfig_750_495.typChannelConfig[3].wCurrentTransformerRatio :=CurrentRatioPQ4;

typConfig_750_495.xWriteConfig := TRUE;
END_ACTION

(* POU 01. PowerQualityMeasurements/PQ_5, FBD *)
PROGRAM PQ_5
VAR
	abProcessImageInput	AT %IW60			: ARRAY[0..23] OF BYTE;
	abProcessImageOutput 	AT %QW68		: ARRAY[0..23] OF BYTE;

	bToken										: BYTE;

	State_750_495 							: Fb_750_495_State;
		typ_750_495_State 						: typ_750_495_State;

	Configuration_750_495					: Fb_750_495_Configuration;
		typConfig_750_495						: typConfig_750_495;
		xReadyConfig								: BOOL;
		bFeedbackConfig							: BYTE;

	AC_Compact_01_750_495				: Fb_750_495_AC_Compact_01;
		rTotalActivePower							: REAL;
		rTotalReactivePower						: REAL;
		rTotalApparentPower						: REAL;
		rTotalPowerFactorPF						: REAL;
		rTotalActiveEnergy							: REAL;
		rTotalReactiveEnergy						: REAL;
		rTotalApparentEnergy						: REAL;
		rCurrentN									: REAL;
		xRotatingField								: BOOL;
		arCurrent									: ARRAY[1..3] OF REAL;
		axOvercurrent								: ARRAY[1..3] OF BOOL;
		arVoltage_L_N							: ARRAY[1..3] OF REAL;
		axUndervoltage							: ARRAY[1..3] OF BOOL;
		axOvervoltage								: ARRAY[1..3] OF BOOL;
		arActivePower								: ARRAY[1..3] OF REAL;
		arReactivePower							: ARRAY[1..3] OF REAL;
		arApparentPower							: ARRAY[1..3] OF REAL;
		arCosPhi									: ARRAY[1..3] OF REAL;
		arPowerFactorPF							: ARRAY[1..3] OF REAL;
		arFrequency								: ARRAY[1..3] OF REAL;
		axNoZero									: ARRAY[1..3] OF BOOL;
		axVoltSag									: ARRAY[1..3] OF BOOL;
		ai4Quadrant								: ARRAY[1..3] OF INT;

		xReadyCompact_01						: BOOL;
		abFeedbackCompact_01					: ARRAY[1..8] OF BYTE;


END_VAR
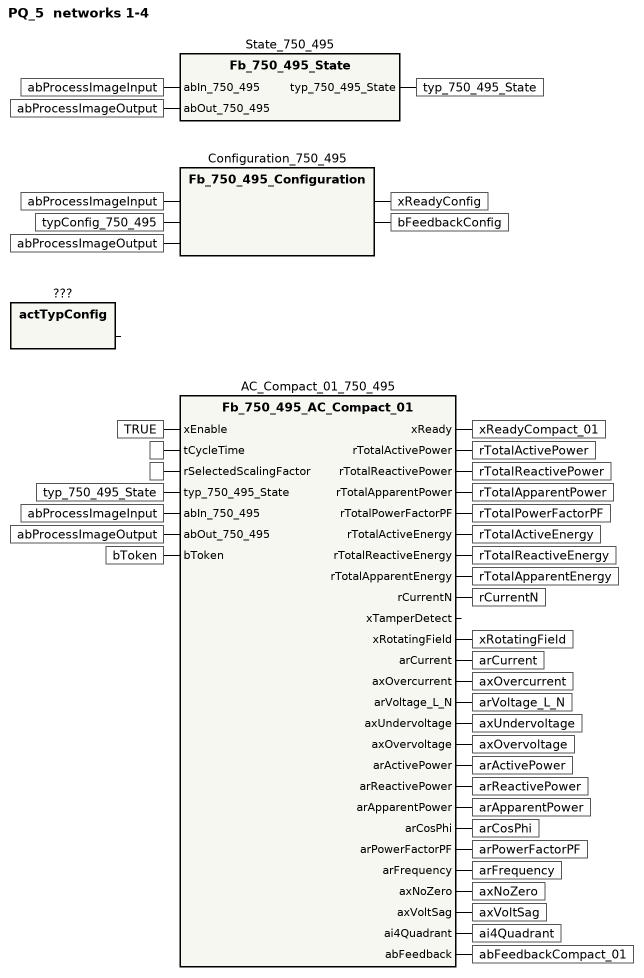
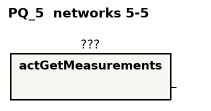
_FBD_ (* Function Block Diagram *)
NETWORK 1
	State_750_495:Fb_750_495_State(abIn_750_495: abProcessImageInput, abOut_750_495: abProcessImageOutput) => typ_750_495_State
NETWORK 2
	Configuration_750_495:Fb_750_495_Configuration(abProcessImageInput, typConfig_750_495, abProcessImageOutput, out 2 => bFeedbackConfig) => xReadyConfig
NETWORK 3
	???:actTypConfig()
NETWORK 4
	AC_Compact_01_750_495:Fb_750_495_AC_Compact_01(xEnable: TRUE, tCycleTime: , rSelectedScalingFactor: , typ_750_495_State: typ_750_495_State, abIn_750_495: abProcessImageInput, abOut_750_495: abProcessImageOutput, bToken: bToken, rTotalActivePower => rTotalActivePower, rTotalReactivePower => rTotalReactivePower, rTotalApparentPower => rTotalApparentPower, rTotalPowerFactorPF => rTotalPowerFactorPF, rTotalActiveEnergy => rTotalActiveEnergy, rTotalReactiveEnergy => rTotalReactiveEnergy, rTotalApparentEnergy => rTotalApparentEnergy, rCurrentN => rCurrentN, xRotatingField => xRotatingField, arCurrent => arCurrent, axOvercurrent => axOvercurrent, arVoltage_L_N => arVoltage_L_N, axUndervoltage => axUndervoltage, axOvervoltage => axOvervoltage, arActivePower => arActivePower, arReactivePower => arReactivePower, arApparentPower => arApparentPower, arCosPhi => arCosPhi, arPowerFactorPF => arPowerFactorPF, arFrequency => arFrequency, axNoZero => axNoZero, axVoltSag => axVoltSag, ai4Quadrant => ai4Quadrant, abFeedback => abFeedbackCompact_01) => xReadyCompact_01
NETWORK 5
	???:actGetMeasurements()
_END_FBD_
(* the same logic as Structured Text *)
(* Network 1 *)
State_750_495(abIn_750_495 := abProcessImageInput, abOut_750_495 := abProcessImageOutput);
typ_750_495_State := State_750_495.typ_750_495_State;
(* Network 2: see the listing above *)
(* Network 3: see the listing above *)
(* Network 4: see the listing above *)
(* Network 5: see the listing above *)
END_PROGRAM
ACTION actGetMeasurements:
arMeasurementsGroup5[1] := arActivePower[1];
arMeasurementsGroup5[2] := arActivePower[2];
arMeasurementsGroup5[3] := arActivePower[3];
arMeasurementsGroup5[4] := arReactivePower[1];
arMeasurementsGroup5[5] := arReactivePower[2];
arMeasurementsGroup5[6] := arReactivePower[3];
arMeasurementsGroup5[7] := arVoltage_L_N[1];
arMeasurementsGroup5[8] := arVoltage_L_N[2];
arMeasurementsGroup5[9] := arVoltage_L_N[3];
arMeasurementsGroup5[10] := arCurrent[1];
arMeasurementsGroup5[11] := arCurrent[2];
arMeasurementsGroup5[12] := arCurrent[3];
arMeasurementsGroup5[13] := arFrequency[1];
arMeasurementsGroup5[14] := arFrequency[2];
arMeasurementsGroup5[15] := arFrequency[3];
arMeasurementsGroup5[16] := rTotalActiveEnergy;
arMeasurementsGroup5[17] := BOOL_TO_REAL(xRotatingField);
arMeasurementsGroup5[18] := rTotalReactiveEnergy;
END_ACTION
ACTION actTypConfig:
typConfig_750_495.typChannelConfig[1].xEnableUserScaling:= TRUE;
typConfig_750_495.typChannelConfig[1].wCurrentTransformerRatio :=CurrentRatioPQ5;

typConfig_750_495.typChannelConfig[2].xEnableUserScaling:= TRUE;
typConfig_750_495.typChannelConfig[2].wCurrentTransformerRatio :=CurrentRatioPQ5;

typConfig_750_495.typChannelConfig[3].xEnableUserScaling:= TRUE;
typConfig_750_495.typChannelConfig[3].wCurrentTransformerRatio :=CurrentRatioPQ5;

typConfig_750_495.xWriteConfig := TRUE;
END_ACTION

(* POU 01. PowerQualityMeasurements/PQ_6, FBD *)
PROGRAM PQ_6
VAR
	abProcessImageInput	AT %IW72			: ARRAY[0..23] OF BYTE;
	abProcessImageOutput 	AT %QW80		: ARRAY[0..23] OF BYTE;

	bToken										: BYTE;

	State_750_495 							: Fb_750_495_State;
		typ_750_495_State 						: typ_750_495_State;

	Configuration_750_495					: Fb_750_495_Configuration;
		typConfig_750_495						: typConfig_750_495;
		xReadyConfig								: BOOL;
		bFeedbackConfig							: BYTE;

	AC_Compact_01_750_495				: Fb_750_495_AC_Compact_01;
		rTotalActivePower							: REAL;
		rTotalReactivePower						: REAL;
		rTotalApparentPower						: REAL;
		rTotalPowerFactorPF						: REAL;
		rTotalActiveEnergy							: REAL;
		rTotalReactiveEnergy						: REAL;
		rTotalApparentEnergy						: REAL;
		rCurrentN									: REAL;
		xRotatingField								: BOOL;
		arCurrent									: ARRAY[1..3] OF REAL;
		axOvercurrent								: ARRAY[1..3] OF BOOL;
		arVoltage_L_N							: ARRAY[1..3] OF REAL;
		axUndervoltage							: ARRAY[1..3] OF BOOL;
		axOvervoltage								: ARRAY[1..3] OF BOOL;
		arActivePower								: ARRAY[1..3] OF REAL;
		arReactivePower							: ARRAY[1..3] OF REAL;
		arApparentPower							: ARRAY[1..3] OF REAL;
		arCosPhi									: ARRAY[1..3] OF REAL;
		arPowerFactorPF							: ARRAY[1..3] OF REAL;
		arFrequency								: ARRAY[1..3] OF REAL;
		axNoZero									: ARRAY[1..3] OF BOOL;
		axVoltSag									: ARRAY[1..3] OF BOOL;
		ai4Quadrant								: ARRAY[1..3] OF INT;

		xReadyCompact_01						: BOOL;
		abFeedbackCompact_01					: ARRAY[1..8] OF BYTE;


END_VAR
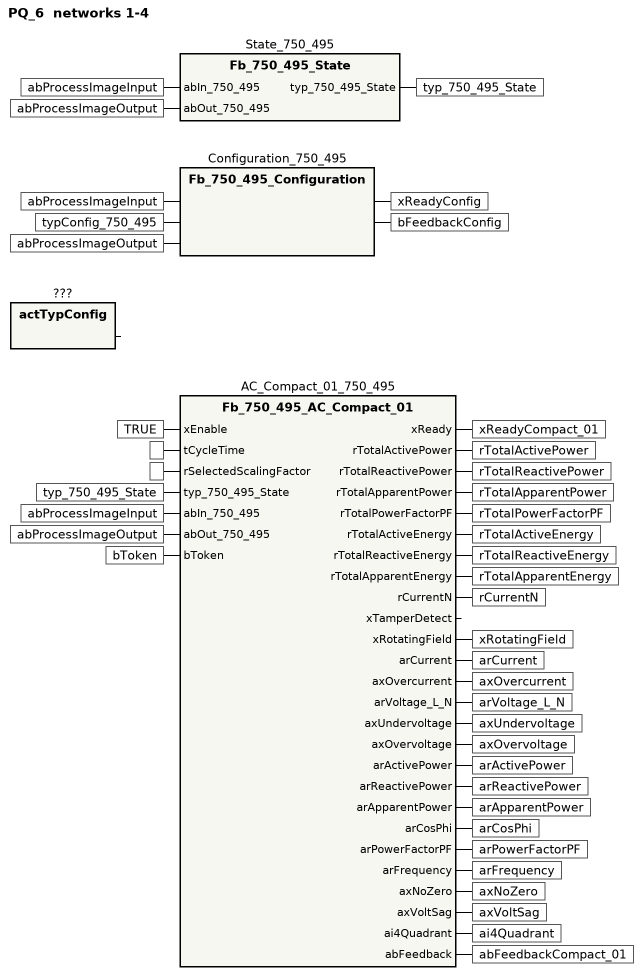
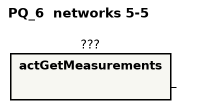
_FBD_ (* Function Block Diagram *)
NETWORK 1
	State_750_495:Fb_750_495_State(abIn_750_495: abProcessImageInput, abOut_750_495: abProcessImageOutput) => typ_750_495_State
NETWORK 2
	Configuration_750_495:Fb_750_495_Configuration(abProcessImageInput, typConfig_750_495, abProcessImageOutput, out 2 => bFeedbackConfig) => xReadyConfig
NETWORK 3
	???:actTypConfig()
NETWORK 4
	AC_Compact_01_750_495:Fb_750_495_AC_Compact_01(xEnable: TRUE, tCycleTime: , rSelectedScalingFactor: , typ_750_495_State: typ_750_495_State, abIn_750_495: abProcessImageInput, abOut_750_495: abProcessImageOutput, bToken: bToken, rTotalActivePower => rTotalActivePower, rTotalReactivePower => rTotalReactivePower, rTotalApparentPower => rTotalApparentPower, rTotalPowerFactorPF => rTotalPowerFactorPF, rTotalActiveEnergy => rTotalActiveEnergy, rTotalReactiveEnergy => rTotalReactiveEnergy, rTotalApparentEnergy => rTotalApparentEnergy, rCurrentN => rCurrentN, xRotatingField => xRotatingField, arCurrent => arCurrent, axOvercurrent => axOvercurrent, arVoltage_L_N => arVoltage_L_N, axUndervoltage => axUndervoltage, axOvervoltage => axOvervoltage, arActivePower => arActivePower, arReactivePower => arReactivePower, arApparentPower => arApparentPower, arCosPhi => arCosPhi, arPowerFactorPF => arPowerFactorPF, arFrequency => arFrequency, axNoZero => axNoZero, axVoltSag => axVoltSag, ai4Quadrant => ai4Quadrant, abFeedback => abFeedbackCompact_01) => xReadyCompact_01
NETWORK 5
	???:actGetMeasurements()
_END_FBD_
(* the same logic as Structured Text *)
(* Network 1 *)
State_750_495(abIn_750_495 := abProcessImageInput, abOut_750_495 := abProcessImageOutput);
typ_750_495_State := State_750_495.typ_750_495_State;
(* Network 2: see the listing above *)
(* Network 3: see the listing above *)
(* Network 4: see the listing above *)
(* Network 5: see the listing above *)
END_PROGRAM
ACTION actGetMeasurements:
arMeasurementsGroup6[1] := arActivePower[1];
arMeasurementsGroup6[2] := arActivePower[2];
arMeasurementsGroup6[3] := arActivePower[3];
arMeasurementsGroup6[4] := arReactivePower[1];
arMeasurementsGroup6[5] := arReactivePower[2];
arMeasurementsGroup6[6] := arReactivePower[3];
arMeasurementsGroup6[7] := arVoltage_L_N[1];
arMeasurementsGroup6[8] := arVoltage_L_N[2];
arMeasurementsGroup6[9] := arVoltage_L_N[3];
arMeasurementsGroup6[10] := arCurrent[1];
arMeasurementsGroup6[11] := arCurrent[2];
arMeasurementsGroup6[12] := arCurrent[3];
arMeasurementsGroup6[13] := arFrequency[1];
arMeasurementsGroup6[14] := arFrequency[2];
arMeasurementsGroup6[15] := arFrequency[3];
arMeasurementsGroup6[16] := rTotalActiveEnergy;
arMeasurementsGroup6[17] := BOOL_TO_REAL(xRotatingField);
arMeasurementsGroup6[18] := rTotalReactiveEnergy;
END_ACTION
ACTION actTypConfig:
typConfig_750_495.typChannelConfig[1].xEnableUserScaling:= TRUE;
typConfig_750_495.typChannelConfig[1].wCurrentTransformerRatio :=CurrentRatioPQ6;

typConfig_750_495.typChannelConfig[2].xEnableUserScaling:= TRUE;
typConfig_750_495.typChannelConfig[2].wCurrentTransformerRatio :=CurrentRatioPQ6;

typConfig_750_495.typChannelConfig[3].xEnableUserScaling:= TRUE;
typConfig_750_495.typChannelConfig[3].wCurrentTransformerRatio :=CurrentRatioPQ6;

typConfig_750_495.xWriteConfig := TRUE;
END_ACTION

(* POU 01. PowerQualityMeasurements/PQ_7, FBD *)
PROGRAM PQ_7
VAR
	abProcessImageInput	AT %IW84			: ARRAY[0..23] OF BYTE;
	abProcessImageOutput 	AT %QW92 			: ARRAY[0..23] OF BYTE;

	bToken										: BYTE;

	State_750_495 							: Fb_750_495_State;
		typ_750_495_State 						: typ_750_495_State;

	Configuration_750_495					: Fb_750_495_Configuration;
		typConfig_750_495						: typConfig_750_495;
		xReadyConfig								: BOOL;
		bFeedbackConfig							: BYTE;

	AC_Compact_01_750_495				: Fb_750_495_AC_Compact_01;
		rTotalActivePower							: REAL;
		rTotalReactivePower						: REAL;
		rTotalApparentPower						: REAL;
		rTotalPowerFactorPF						: REAL;
		rTotalActiveEnergy							: REAL;
		rTotalReactiveEnergy						: REAL;
		rTotalApparentEnergy						: REAL;
		rCurrentN									: REAL;
		xRotatingField								: BOOL;
		arCurrent									: ARRAY[1..3] OF REAL;
		axOvercurrent								: ARRAY[1..3] OF BOOL;
		arVoltage_L_N							: ARRAY[1..3] OF REAL;
		axUndervoltage							: ARRAY[1..3] OF BOOL;
		axOvervoltage								: ARRAY[1..3] OF BOOL;
		arActivePower								: ARRAY[1..3] OF REAL;
		arReactivePower							: ARRAY[1..3] OF REAL;
		arApparentPower							: ARRAY[1..3] OF REAL;
		arCosPhi									: ARRAY[1..3] OF REAL;
		arPowerFactorPF							: ARRAY[1..3] OF REAL;
		arFrequency								: ARRAY[1..3] OF REAL;
		axNoZero									: ARRAY[1..3] OF BOOL;
		axVoltSag									: ARRAY[1..3] OF BOOL;
		ai4Quadrant								: ARRAY[1..3] OF INT;

		xReadyCompact_01						: BOOL;
		abFeedbackCompact_01					: ARRAY[1..8] OF BYTE;


END_VAR
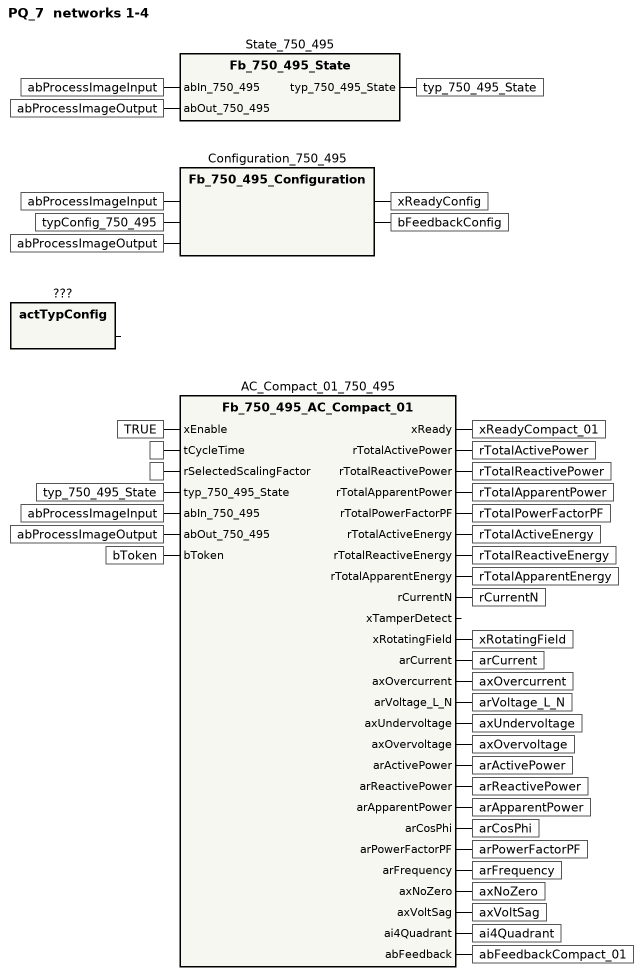
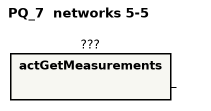
_FBD_ (* Function Block Diagram *)
NETWORK 1
	State_750_495:Fb_750_495_State(abIn_750_495: abProcessImageInput, abOut_750_495: abProcessImageOutput) => typ_750_495_State
NETWORK 2
	Configuration_750_495:Fb_750_495_Configuration(abProcessImageInput, typConfig_750_495, abProcessImageOutput, out 2 => bFeedbackConfig) => xReadyConfig
NETWORK 3
	???:actTypConfig()
NETWORK 4
	AC_Compact_01_750_495:Fb_750_495_AC_Compact_01(xEnable: TRUE, tCycleTime: , rSelectedScalingFactor: , typ_750_495_State: typ_750_495_State, abIn_750_495: abProcessImageInput, abOut_750_495: abProcessImageOutput, bToken: bToken, rTotalActivePower => rTotalActivePower, rTotalReactivePower => rTotalReactivePower, rTotalApparentPower => rTotalApparentPower, rTotalPowerFactorPF => rTotalPowerFactorPF, rTotalActiveEnergy => rTotalActiveEnergy, rTotalReactiveEnergy => rTotalReactiveEnergy, rTotalApparentEnergy => rTotalApparentEnergy, rCurrentN => rCurrentN, xRotatingField => xRotatingField, arCurrent => arCurrent, axOvercurrent => axOvercurrent, arVoltage_L_N => arVoltage_L_N, axUndervoltage => axUndervoltage, axOvervoltage => axOvervoltage, arActivePower => arActivePower, arReactivePower => arReactivePower, arApparentPower => arApparentPower, arCosPhi => arCosPhi, arPowerFactorPF => arPowerFactorPF, arFrequency => arFrequency, axNoZero => axNoZero, axVoltSag => axVoltSag, ai4Quadrant => ai4Quadrant, abFeedback => abFeedbackCompact_01) => xReadyCompact_01
NETWORK 5
	???:actGetMeasurements()
_END_FBD_
(* the same logic as Structured Text *)
(* Network 1 *)
State_750_495(abIn_750_495 := abProcessImageInput, abOut_750_495 := abProcessImageOutput);
typ_750_495_State := State_750_495.typ_750_495_State;
(* Network 2: see the listing above *)
(* Network 3: see the listing above *)
(* Network 4: see the listing above *)
(* Network 5: see the listing above *)
END_PROGRAM
ACTION actGetMeasurements:
arMeasurementsGroup7[1] := arActivePower[1];
arMeasurementsGroup7[2] := arActivePower[2];
arMeasurementsGroup7[3] := arActivePower[3];
arMeasurementsGroup7[4] := arReactivePower[1];
arMeasurementsGroup7[5] := arReactivePower[2];
arMeasurementsGroup7[6] := arReactivePower[3];
arMeasurementsGroup7[7] := arVoltage_L_N[1];
arMeasurementsGroup7[8] := arVoltage_L_N[2];
arMeasurementsGroup7[9] := arVoltage_L_N[3];
arMeasurementsGroup7[10] := arCurrent[1];
arMeasurementsGroup7[11] := arCurrent[2];
arMeasurementsGroup7[12] := arCurrent[3];
arMeasurementsGroup7[13] := arFrequency[1];
arMeasurementsGroup7[14] := arFrequency[2];
arMeasurementsGroup7[15] := arFrequency[3];
arMeasurementsGroup7[16] := rTotalActiveEnergy;
arMeasurementsGroup7[17] := BOOL_TO_REAL(xRotatingField);
arMeasurementsGroup7[18] := rTotalReactiveEnergy;
END_ACTION
ACTION actTypConfig:
typConfig_750_495.typChannelConfig[1].xEnableUserScaling:= TRUE;
typConfig_750_495.typChannelConfig[1].wCurrentTransformerRatio :=CurrentRatioPQ7;

typConfig_750_495.typChannelConfig[2].xEnableUserScaling:= TRUE;
typConfig_750_495.typChannelConfig[2].wCurrentTransformerRatio :=CurrentRatioPQ7;

typConfig_750_495.typChannelConfig[3].xEnableUserScaling:= TRUE;
typConfig_750_495.typChannelConfig[3].wCurrentTransformerRatio :=CurrentRatioPQ7;

typConfig_750_495.xWriteConfig := TRUE;
END_ACTION

(* POU 01. PowerQualityMeasurements/PQ_8, FBD *)
PROGRAM PQ_8
VAR
	abProcessImageInput	AT %IW96			: ARRAY[0..23] OF BYTE;
	abProcessImageOutput 	AT %QW104 		: ARRAY[0..23] OF BYTE;

	bToken										: BYTE;

	State_750_495 							: Fb_750_495_State;
		typ_750_495_State 						: typ_750_495_State;

	Configuration_750_495					: Fb_750_495_Configuration;
		typConfig_750_495						: typConfig_750_495;
		xReadyConfig								: BOOL;
		bFeedbackConfig							: BYTE;

	AC_Compact_01_750_495				: Fb_750_495_AC_Compact_01;
		rTotalActivePower							: REAL;
		rTotalReactivePower						: REAL;
		rTotalApparentPower						: REAL;
		rTotalPowerFactorPF						: REAL;
		rTotalActiveEnergy							: REAL;
		rTotalReactiveEnergy						: REAL;
		rTotalApparentEnergy						: REAL;
		rCurrentN									: REAL;
		xRotatingField								: BOOL;
		arCurrent									: ARRAY[1..3] OF REAL;
		axOvercurrent								: ARRAY[1..3] OF BOOL;
		arVoltage_L_N							: ARRAY[1..3] OF REAL;
		axUndervoltage							: ARRAY[1..3] OF BOOL;
		axOvervoltage								: ARRAY[1..3] OF BOOL;
		arActivePower								: ARRAY[1..3] OF REAL;
		arReactivePower							: ARRAY[1..3] OF REAL;
		arApparentPower							: ARRAY[1..3] OF REAL;
		arCosPhi									: ARRAY[1..3] OF REAL;
		arPowerFactorPF							: ARRAY[1..3] OF REAL;
		arFrequency								: ARRAY[1..3] OF REAL;
		axNoZero									: ARRAY[1..3] OF BOOL;
		axVoltSag									: ARRAY[1..3] OF BOOL;
		ai4Quadrant								: ARRAY[1..3] OF INT;

		xReadyCompact_01						: BOOL;
		abFeedbackCompact_01					: ARRAY[1..8] OF BYTE;


END_VAR
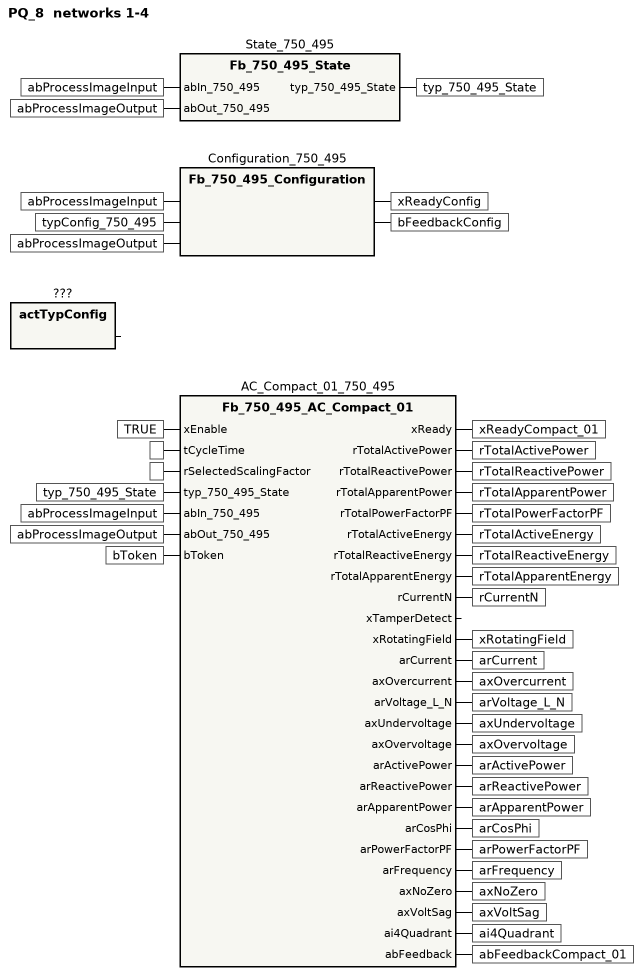
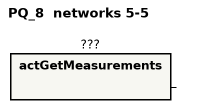
_FBD_ (* Function Block Diagram *)
NETWORK 1
	State_750_495:Fb_750_495_State(abIn_750_495: abProcessImageInput, abOut_750_495: abProcessImageOutput) => typ_750_495_State
NETWORK 2
	Configuration_750_495:Fb_750_495_Configuration(abProcessImageInput, typConfig_750_495, abProcessImageOutput, out 2 => bFeedbackConfig) => xReadyConfig
NETWORK 3
	???:actTypConfig()
NETWORK 4
	AC_Compact_01_750_495:Fb_750_495_AC_Compact_01(xEnable: TRUE, tCycleTime: , rSelectedScalingFactor: , typ_750_495_State: typ_750_495_State, abIn_750_495: abProcessImageInput, abOut_750_495: abProcessImageOutput, bToken: bToken, rTotalActivePower => rTotalActivePower, rTotalReactivePower => rTotalReactivePower, rTotalApparentPower => rTotalApparentPower, rTotalPowerFactorPF => rTotalPowerFactorPF, rTotalActiveEnergy => rTotalActiveEnergy, rTotalReactiveEnergy => rTotalReactiveEnergy, rTotalApparentEnergy => rTotalApparentEnergy, rCurrentN => rCurrentN, xRotatingField => xRotatingField, arCurrent => arCurrent, axOvercurrent => axOvercurrent, arVoltage_L_N => arVoltage_L_N, axUndervoltage => axUndervoltage, axOvervoltage => axOvervoltage, arActivePower => arActivePower, arReactivePower => arReactivePower, arApparentPower => arApparentPower, arCosPhi => arCosPhi, arPowerFactorPF => arPowerFactorPF, arFrequency => arFrequency, axNoZero => axNoZero, axVoltSag => axVoltSag, ai4Quadrant => ai4Quadrant, abFeedback => abFeedbackCompact_01) => xReadyCompact_01
NETWORK 5
	???:actGetMeasurements()
_END_FBD_
(* the same logic as Structured Text *)
(* Network 1 *)
State_750_495(abIn_750_495 := abProcessImageInput, abOut_750_495 := abProcessImageOutput);
typ_750_495_State := State_750_495.typ_750_495_State;
(* Network 2: see the listing above *)
(* Network 3: see the listing above *)
(* Network 4: see the listing above *)
(* Network 5: see the listing above *)
END_PROGRAM
ACTION actGetMeasurements:
arMeasurementsGroup8[1] := arActivePower[1];
arMeasurementsGroup8[2] := arActivePower[2];
arMeasurementsGroup8[3] := arActivePower[3];
arMeasurementsGroup8[4] := arReactivePower[1];
arMeasurementsGroup8[5] := arReactivePower[2];
arMeasurementsGroup8[6] := arReactivePower[3];
arMeasurementsGroup8[7] := arVoltage_L_N[1];
arMeasurementsGroup8[8] := arVoltage_L_N[2];
arMeasurementsGroup8[9] := arVoltage_L_N[3];
arMeasurementsGroup8[10] := arCurrent[1];
arMeasurementsGroup8[11] := arCurrent[2];
arMeasurementsGroup8[12] := arCurrent[3];
arMeasurementsGroup8[13] := arFrequency[1];
arMeasurementsGroup8[14] := arFrequency[2];
arMeasurementsGroup8[15] := arFrequency[3];
arMeasurementsGroup8[16] := rTotalActiveEnergy;
arMeasurementsGroup8[17] := BOOL_TO_REAL(xRotatingField);
arMeasurementsGroup8[18] := rTotalReactiveEnergy;
END_ACTION
ACTION actTypConfig:
typConfig_750_495.typChannelConfig[1].xEnableUserScaling:= TRUE;
typConfig_750_495.typChannelConfig[1].wCurrentTransformerRatio :=CurrentRatioPQ8;

typConfig_750_495.typChannelConfig[2].xEnableUserScaling:= TRUE;
typConfig_750_495.typChannelConfig[2].wCurrentTransformerRatio :=CurrentRatioPQ8;

typConfig_750_495.typChannelConfig[3].xEnableUserScaling:= TRUE;
typConfig_750_495.typChannelConfig[3].wCurrentTransformerRatio :=CurrentRatioPQ8;

typConfig_750_495.xWriteConfig := TRUE;
END_ACTION

(* POU 01. PowerQualityMeasurements/PQ_9, FBD *)
PROGRAM PQ_9
VAR
	abProcessImageInput	AT %IW108		: ARRAY[0..23] OF BYTE;
	abProcessImageOutput 	AT %QW116		: ARRAY[0..23] OF BYTE;

	bToken										: BYTE;

	State_750_495 							: Fb_750_495_State;
		typ_750_495_State 						: typ_750_495_State;

	Configuration_750_495					: Fb_750_495_Configuration;
		typConfig_750_495						: typConfig_750_495;
		xReadyConfig								: BOOL;
		bFeedbackConfig							: BYTE;

	AC_Compact_01_750_495				: Fb_750_495_AC_Compact_01;
		rTotalActivePower							: REAL;
		rTotalReactivePower						: REAL;
		rTotalApparentPower						: REAL;
		rTotalPowerFactorPF						: REAL;
		rTotalActiveEnergy							: REAL;
		rTotalReactiveEnergy						: REAL;
		rTotalApparentEnergy						: REAL;
		rCurrentN									: REAL;
		xRotatingField								: BOOL;
		arCurrent									: ARRAY[1..3] OF REAL;
		axOvercurrent								: ARRAY[1..3] OF BOOL;
		arVoltage_L_N							: ARRAY[1..3] OF REAL;
		axUndervoltage							: ARRAY[1..3] OF BOOL;
		axOvervoltage								: ARRAY[1..3] OF BOOL;
		arActivePower								: ARRAY[1..3] OF REAL;
		arReactivePower							: ARRAY[1..3] OF REAL;
		arApparentPower							: ARRAY[1..3] OF REAL;
		arCosPhi									: ARRAY[1..3] OF REAL;
		arPowerFactorPF							: ARRAY[1..3] OF REAL;
		arFrequency								: ARRAY[1..3] OF REAL;
		axNoZero									: ARRAY[1..3] OF BOOL;
		axVoltSag									: ARRAY[1..3] OF BOOL;
		ai4Quadrant								: ARRAY[1..3] OF INT;

		xReadyCompact_01						: BOOL;
		abFeedbackCompact_01					: ARRAY[1..8] OF BYTE;


END_VAR
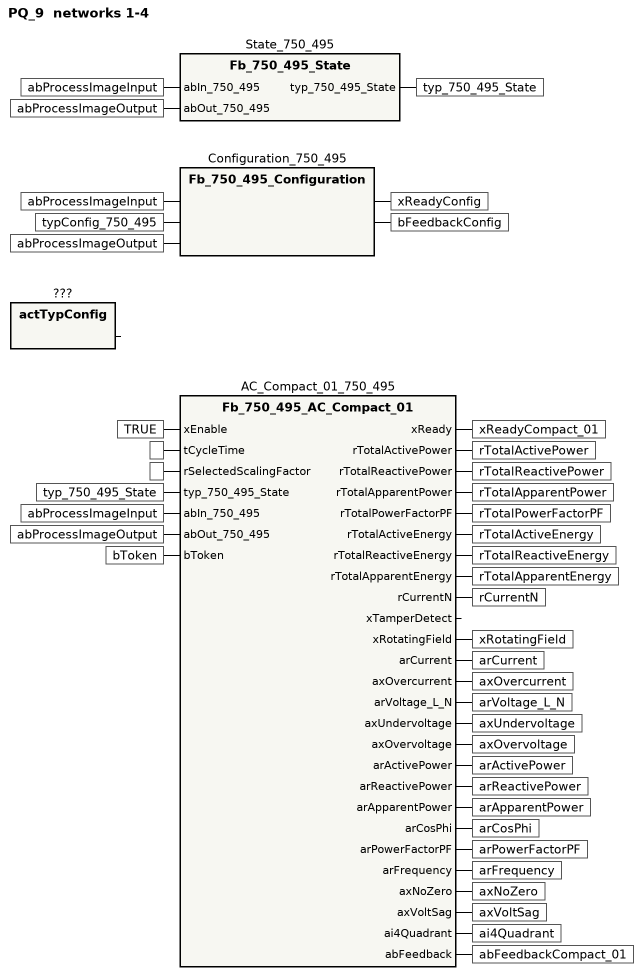
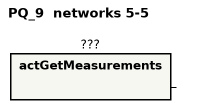
_FBD_ (* Function Block Diagram *)
NETWORK 1
	State_750_495:Fb_750_495_State(abIn_750_495: abProcessImageInput, abOut_750_495: abProcessImageOutput) => typ_750_495_State
NETWORK 2
	Configuration_750_495:Fb_750_495_Configuration(abProcessImageInput, typConfig_750_495, abProcessImageOutput, out 2 => bFeedbackConfig) => xReadyConfig
NETWORK 3
	???:actTypConfig()
NETWORK 4
	AC_Compact_01_750_495:Fb_750_495_AC_Compact_01(xEnable: TRUE, tCycleTime: , rSelectedScalingFactor: , typ_750_495_State: typ_750_495_State, abIn_750_495: abProcessImageInput, abOut_750_495: abProcessImageOutput, bToken: bToken, rTotalActivePower => rTotalActivePower, rTotalReactivePower => rTotalReactivePower, rTotalApparentPower => rTotalApparentPower, rTotalPowerFactorPF => rTotalPowerFactorPF, rTotalActiveEnergy => rTotalActiveEnergy, rTotalReactiveEnergy => rTotalReactiveEnergy, rTotalApparentEnergy => rTotalApparentEnergy, rCurrentN => rCurrentN, xRotatingField => xRotatingField, arCurrent => arCurrent, axOvercurrent => axOvercurrent, arVoltage_L_N => arVoltage_L_N, axUndervoltage => axUndervoltage, axOvervoltage => axOvervoltage, arActivePower => arActivePower, arReactivePower => arReactivePower, arApparentPower => arApparentPower, arCosPhi => arCosPhi, arPowerFactorPF => arPowerFactorPF, arFrequency => arFrequency, axNoZero => axNoZero, axVoltSag => axVoltSag, ai4Quadrant => ai4Quadrant, abFeedback => abFeedbackCompact_01) => xReadyCompact_01
NETWORK 5
	???:actGetMeasurements()
_END_FBD_
(* the same logic as Structured Text *)
(* Network 1 *)
State_750_495(abIn_750_495 := abProcessImageInput, abOut_750_495 := abProcessImageOutput);
typ_750_495_State := State_750_495.typ_750_495_State;
(* Network 2: see the listing above *)
(* Network 3: see the listing above *)
(* Network 4: see the listing above *)
(* Network 5: see the listing above *)
END_PROGRAM
ACTION actGetMeasurements:
arMeasurementsGroup9[1] := arActivePower[1];
arMeasurementsGroup9[2] := arActivePower[2];
arMeasurementsGroup9[3] := arActivePower[3];
arMeasurementsGroup9[4] := arReactivePower[1];
arMeasurementsGroup9[5] := arReactivePower[2];
arMeasurementsGroup9[6] := arReactivePower[3];
arMeasurementsGroup9[7] := arVoltage_L_N[1];
arMeasurementsGroup9[8] := arVoltage_L_N[2];
arMeasurementsGroup9[9] := arVoltage_L_N[3];
arMeasurementsGroup9[10] := arCurrent[1];
arMeasurementsGroup9[11] := arCurrent[2];
arMeasurementsGroup9[12] := arCurrent[3];
arMeasurementsGroup9[13] := arFrequency[1];
arMeasurementsGroup9[14] := arFrequency[2];
arMeasurementsGroup9[15] := arFrequency[3];
arMeasurementsGroup9[16] := rTotalActiveEnergy;
arMeasurementsGroup9[17] := BOOL_TO_REAL(xRotatingField);
arMeasurementsGroup9[18] := rTotalReactiveEnergy;
END_ACTION
ACTION actTypConfig:
typConfig_750_495.typChannelConfig[1].xEnableUserScaling:= TRUE;
typConfig_750_495.typChannelConfig[1].wCurrentTransformerRatio :=CurrentRatioPQ9;

typConfig_750_495.typChannelConfig[2].xEnableUserScaling:= TRUE;
typConfig_750_495.typChannelConfig[2].wCurrentTransformerRatio :=CurrentRatioPQ9;

typConfig_750_495.typChannelConfig[3].xEnableUserScaling:= TRUE;
typConfig_750_495.typChannelConfig[3].wCurrentTransformerRatio :=CurrentRatioPQ9;

typConfig_750_495.xWriteConfig := TRUE;
END_ACTION

(* POU 05. Modbus System State Array/variables_to_system_array, ST *)
PROGRAM variables_to_system_array
VAR
	i: INT;
	j: INT;
	start : INT;
END_VAR
(* https://docs.google.com/spreadsheets/d/1TR7oXGZyEmNnGigmreKdtnpXsz8mxFcoB4b4beNITCA/edit *)

(* loop trough all variable and measurements groups *)
FOR j := 0 TO iNumberMeasurementGroups-1 DO

	start := j*iNumberMeasurementVar;
	FOR i := 1 TO iNumberMeasurementVar-1  DO

		IF i +start <= iNumberMeasurementVar THEN
			arSystemState[i+start] := arMeasurementsGroupA[i];
		END_IF

		IF i +start > iNumberMeasurementVar AND  i +start <= 2*iNumberMeasurementVar THEN
			arSystemState[i+start] := arMeasurementsGroupB[i];
		END_IF

		IF i +start > 2*iNumberMeasurementVar AND  i +start <= 3*iNumberMeasurementVar THEN
			arSystemState[i+start] := arMeasurementsGroup1[i];
		END_IF

		IF i +start > 3*iNumberMeasurementVar AND  i +start <= 4*iNumberMeasurementVar THEN
			arSystemState[i+start] := arMeasurementsGroup2[i];
		END_IF

		IF i +start > 4*iNumberMeasurementVar AND  i +start <= 5*iNumberMeasurementVar THEN
			arSystemState[i+start] := arMeasurementsGroup3[i];
		END_IF

		IF i +start > 5*iNumberMeasurementVar AND  i +start <= 6*iNumberMeasurementVar THEN
			arSystemState[i+start] := arMeasurementsGroup4[i];
		END_IF

		IF i +start > 6*iNumberMeasurementVar AND  i +start <= 7*iNumberMeasurementVar THEN
			arSystemState[i+start] := arMeasurementsGroup5[i];
		END_IF
		IF i +start > 7*iNumberMeasurementVar AND  i +start <= 8*iNumberMeasurementVar THEN
			arSystemState[i+start] := arMeasurementsGroup6[i];
		END_IF

		IF i +start > 8*iNumberMeasurementVar AND  i +start <= 9*iNumberMeasurementVar THEN
			arSystemState[i+start] := arMeasurementsGroup7[i];
		END_IF

		IF i +start > 9*iNumberMeasurementVar AND  i +start <= 10*iNumberMeasurementVar THEN
			arSystemState[i+start] := arMeasurementsGroup8[i];
		END_IF

		IF i +start > 10*iNumberMeasurementVar AND  i +start <= 11*iNumberMeasurementVar THEN
			arSystemState[i+start] := arMeasurementsGroup9[i];
		END_IF

	END_FOR
END_FOR

(* _____ ALWAYS UDPATE (REVERSRE) THE WRITABLE MODBUS PARAMETERS _____

Bus_Connector_3F_Sync_close_requested_modbus 					: BOOL;
Bus_Connector_3F_Sync_denied_modbus				 				: BOOL;
example:
	Bus_Connector_3F_Sync_close_requested_modbus:=REAL_TO_BOOL(arSystemState[219]);
	Bus_Connector_3F_Sync_denied_modbus :=REAL_TO_BOOL(arSystemState[220]);
*)

(* other system variable*)
arSystemState[199] :=Bus_Connector_L1_P;
arSystemState[200] :=Bus_Connector_L2_P;
arSystemState[201] :=Bus_Connector_L3_P;
arSystemState[202] :=Bus_Connector_L1_Q;
arSystemState[203] :=Bus_Connector_L2_Q;
arSystemState[204] :=Bus_Connector_L3_Q;
arSystemState[205] :=Bus_Connector_L1_V;
arSystemState[206] :=Bus_Connector_L2_V;
arSystemState[207] :=Bus_Connector_L3_V;
arSystemState[208] :=Bus_Connector_L1_I;
arSystemState[209] :=Bus_Connector_L2_I;
arSystemState[210] :=Bus_Connector_L3_I;
arSystemState[211] :=Bus_Connector_L1_f;
arSystemState[212] :=Bus_Connector_L2_f;
arSystemState[213] :=Bus_Connector_L3_f;
arSystemState[214] :=Bus_Connector_3F_CosPhi;
arSystemState[215] :=BOOL_TO_REAL(Bus_Connector_3F_Sync_close_requested);
arSystemState[216] :=BOOL_TO_REAL(Bus_Connector_3F_Sync_closed);
arSystemState[217] :=BOOL_TO_REAL(Bus_Connector_3F_Sync_close_requested_panel);
arSystemState[218] :=BOOL_TO_REAL(Bus_Connector_3F_Sync_denied_panel);
Bus_Connector_3F_Sync_close_requested_modbus := REAL_TO_BOOL(arSystemState[219]);
Bus_Connector_3F_Sync_denied_modbus := REAL_TO_BOOL(arSystemState[220]);
arSystemState[221] :=Bus_Connector_3F_Field_Rotation;
(*arSystemState[222] :=BOOL_TO_REAL(CHP_control_grid_bus_select_controlswitch);
arSystemState[223] :=BOOL_TO_REAL(CHP_control_baterry_bus_select_controlswitch);
arSystemState[224] :=BOOL_TO_REAL(CHP_control_auto_bus_select_controlswitch);*)
arSystemState[225] :=BOOL_TO_REAL(CHP_control_Offgrid_request);
arSystemState[226] :=CHP_control_Offgrid_Active_Power_control;
arSystemState[227] :=BOOL_TO_REAL(CHP_control_internal_contacter_switch_state);
arSystemState[228] :=EV_control_control_signal;
arSystemState[229] :=Mixer1_control_control_signal;
arSystemState[230] :=BOOL_TO_REAL(Group1_3F_Auto_relay_control_battery_bus);
arSystemState[231] :=BOOL_TO_REAL(Group1_3F_Auto_relay_control_grid_bus);
arSystemState[232] :=BOOL_TO_REAL(Group1_3F_Selector_auto_bus_select);
arSystemState[233] :=BOOL_TO_REAL(Group1_3F_relay_state_battery_bus);
arSystemState[234] :=BOOL_TO_REAL(Group1_3F_relay_state_grid_bus);
arSystemState[235] :=BOOL_TO_REAL(Group2_3F_Auto_relay_control_battery_bus);
arSystemState[236] :=BOOL_TO_REAL(Group2_3F_Auto_relay_control_grid_bus);
arSystemState[237] :=BOOL_TO_REAL(Group2_3F_Selector_auto_bus_select);
arSystemState[238] :=BOOL_TO_REAL(Group2_3F_relay_state_battery_bus);
arSystemState[239] :=BOOL_TO_REAL(Group2_3F_relay_state_grid_bus);
arSystemState[240] :=BOOL_TO_REAL(Group3_3F_Auto_relay_control_battery_bus);
arSystemState[241] :=BOOL_TO_REAL(Group3_3F_Auto_relay_control_grid_bus);
arSystemState[242] :=BOOL_TO_REAL(Group3_3F_Selector_auto_bus_select);
arSystemState[243] :=BOOL_TO_REAL(Group3_3F_relay_state_battery_bus);
arSystemState[244] :=BOOL_TO_REAL(Group3_3F_relay_state_grid_bus);
arSystemState[245] :=BOOL_TO_REAL(Group4_3F_Auto_relay_control_battery_bus);
arSystemState[246] :=BOOL_TO_REAL(Group4_3F_Auto_relay_control_grid_bus);
arSystemState[247] :=BOOL_TO_REAL(Group4_3F_Selector_auto_bus_select);
arSystemState[248] :=BOOL_TO_REAL(Group4_3F_relay_state_battery_bus);
arSystemState[249] :=BOOL_TO_REAL(Group4_3F_relay_state_grid_bus);
arSystemState[250] :=BOOL_TO_REAL(Group5_3F_Auto_relay_control_battery_bus);
arSystemState[251] :=BOOL_TO_REAL(Group5_3F_Auto_relay_control_grid_bus);
arSystemState[252] :=BOOL_TO_REAL(Group5_3F_Selector_auto_bus_select);
arSystemState[253] :=BOOL_TO_REAL(Group5_3F_relay_state_battery_bus);
arSystemState[254] :=BOOL_TO_REAL(Group5_3F_relay_state_grid_bus);
arSystemState[255] :=BOOL_TO_REAL(Group6_3F_Auto_relay_control_battery_bus);
arSystemState[256] :=BOOL_TO_REAL(Group6_3F_Auto_relay_control_grid_bus);
arSystemState[257] :=BOOL_TO_REAL(Group6_3F_Selector_auto_bus_select);
arSystemState[258] :=BOOL_TO_REAL(Group6_3F_relay_state_battery_bus);
arSystemState[259] :=BOOL_TO_REAL(Group6_3F_relay_state_grid_bus);
arSystemState[260] :=BOOL_TO_REAL(Group7_3F_Auto_relay_control_battery_bus);
arSystemState[261] :=BOOL_TO_REAL(Group7_3F_Auto_relay_control_grid_bus);
arSystemState[262] :=BOOL_TO_REAL(Group7_3F_Selector_auto_bus_select);
arSystemState[263] :=BOOL_TO_REAL(Group7_3F_relay_state_battery_bus);
arSystemState[264] :=BOOL_TO_REAL(Group7_3F_relay_state_grid_bus);
arSystemState[265] :=BOOL_TO_REAL(Group8_3F_Auto_relay_control_battery_bus);
arSystemState[266] :=BOOL_TO_REAL(Group8_3F_Auto_relay_control_grid_bus);
arSystemState[267] :=BOOL_TO_REAL(Group8_3F_Selector_auto_bus_select);
arSystemState[268] :=BOOL_TO_REAL(Group8_3F_relay_state_battery_bus);
arSystemState[269] :=BOOL_TO_REAL(Group8_3F_relay_state_grid_bus);
arSystemState[270] :=BOOL_TO_REAL(Group9_3F_Auto_relay_control_battery_bus);
arSystemState[271] :=BOOL_TO_REAL(Group9_3F_Auto_relay_control_grid_bus);
arSystemState[272] :=BOOL_TO_REAL(Group9_3F_Selector_auto_bus_select);
arSystemState[273] :=BOOL_TO_REAL(Group9_3F_relay_state_battery_bus);
arSystemState[274] :=BOOL_TO_REAL(Group9_3F_relay_state_grid_bus);

IF Group_control_Frequencybased_parameters_initialized = FALSE THEN
arSystemState[275] :=BOOL_TO_REAL(Group_control_Frequencybased_bus_selecting_state);
arSystemState[276] :=Group_control_min_time_above_switch_frequency;
arSystemState[277] :=Group_control_min_time_below_switch_frequency;
arSystemState[278] :=Group1_3F_Switch_frequency_to_batterybus;
arSystemState[279] :=Group1_3F_Switch_frequency_to_gridbus;
arSystemState[280] :=Group1_3F_min_time_between_switching;
arSystemState[281] :=Group2_3F_Switch_frequency_to_batterybus;
arSystemState[282] :=Group2_3F_Switch_frequency_to_gridbus;
arSystemState[283] :=Group2_3F_min_time_between_switching;
arSystemState[284] :=Group3_3F_Switch_frequency_to_batterybus;
arSystemState[285] :=Group3_3F_Switch_frequency_to_gridbus;
arSystemState[286] :=Group3_3F_min_time_between_switching;
arSystemState[287] :=Group4_3F_Switch_frequency_to_batterybus;
arSystemState[288] :=Group4_3F_Switch_frequency_to_gridbus;
arSystemState[289] :=Group4_3F_min_time_between_switching;
arSystemState[290] :=Group5_3F_Switch_frequency_to_batterybus;

arSystemState[291] :=Group5_3F_Switch_frequency_to_gridbus;
arSystemState[292] :=Group5_3F_min_time_between_switching;
arSystemState[293] :=Group6_3F_Switch_frequency_to_batterybus;
arSystemState[294] :=Group6_3F_Switch_frequency_to_gridbus;
arSystemState[295] :=Group6_3F_min_time_between_switching;
arSystemState[296] :=Group7_3F_Switch_frequency_to_batterybus;
arSystemState[297] :=Group7_3F_Switch_frequency_to_gridbus;
arSystemState[298] :=Group7_3F_min_time_between_switching;
arSystemState[299] :=Group8_3F_Switch_frequency_to_batterybus;
arSystemState[300] :=Group8_3F_Switch_frequency_to_gridbus;
arSystemState[301] :=Group8_3F_min_time_between_switching;
arSystemState[302] :=Group9_3F_Switch_frequency_to_batterybus;
arSystemState[303] :=Group9_3F_Switch_frequency_to_gridbus;
arSystemState[304] :=Group9_3F_min_time_between_switching;
Group_control_Frequencybased_parameters_initialized := TRUE;
ELSE
Group_control_Frequencybased_bus_selecting_state := REAL_TO_BOOL(arSystemState[275]);
Group_control_min_time_above_switch_frequency := arSystemState[276];
Group_control_min_time_below_switch_frequency := arSystemState[277];
Group1_3F_Switch_frequency_to_batterybus := arSystemState[278];
Group1_3F_Switch_frequency_to_gridbus := arSystemState[279];
Group1_3F_min_time_between_switching := arSystemState[280];
Group2_3F_Switch_frequency_to_batterybus := arSystemState[281];
Group2_3F_Switch_frequency_to_gridbus := arSystemState[282];
Group2_3F_min_time_between_switching := arSystemState[283];
Group3_3F_Switch_frequency_to_batterybus := arSystemState[284];
Group3_3F_Switch_frequency_to_gridbus := arSystemState[285];
Group3_3F_min_time_between_switching := arSystemState[286];
Group4_3F_Switch_frequency_to_batterybus := arSystemState[287];
Group4_3F_Switch_frequency_to_gridbus := arSystemState[288];
Group4_3F_min_time_between_switching := arSystemState[289];
Group5_3F_Switch_frequency_to_batterybus := arSystemState[290];
Group5_3F_Switch_frequency_to_gridbus := arSystemState[291];
Group5_3F_min_time_between_switching := arSystemState[292];
Group6_3F_Switch_frequency_to_batterybus := arSystemState[293];
Group6_3F_Switch_frequency_to_gridbus := arSystemState[294];
Group6_3F_min_time_between_switching := arSystemState[295];
Group7_3F_Switch_frequency_to_batterybus := arSystemState[296];
Group7_3F_Switch_frequency_to_gridbus := arSystemState[297];
Group7_3F_min_time_between_switching := arSystemState[298];
Group8_3F_Switch_frequency_to_batterybus := arSystemState[299];
Group8_3F_Switch_frequency_to_gridbus := arSystemState[300];
Group8_3F_min_time_between_switching := arSystemState[301];
Group9_3F_Switch_frequency_to_batterybus := arSystemState[302];
Group9_3F_Switch_frequency_to_gridbus := arSystemState[303];
Group9_3F_min_time_between_switching := arSystemState[304];
END_IF;
arSystemState[305] :=BOOL_TO_REAL(Control_panel_status_warning_led);
arSystemState[306] :=BOOL_TO_REAL(Control_panel_status_error_led);
arSystemState[307] :=BOOL_TO_REAL(Control_panel_status_operational_led);

(* REGISTERS FOR THE ALFEN BATTERY*)
TheBattery_SOC_real := arSystemState[308];
TheBattery_SOC_simulated := arSystemState[309];
arSystemState[310] :=TheBattery_bool_use_PLC_SOC;
arSystemState[311] :=TheBattery_SOC_PLC_SOC_setpoint;
END_PROGRAM

(* POU 02. Batterybus Frequency to Analog Out/CHP_Controller, FBD *)
PROGRAM CHP_Controller
(*CHP_control_Offgrid_Active_Power_control  range:
CHP_control_Offgrid_Active_Power_control = Word 0 equals 4mA output, giving 60kW
CHP_control_Offgrid_Active_Power_control = Word 32767 equals 20mA output, giving 120kW*)
VAR
	RAMP_REAL: RAMP_REAL;
	Frequency_to_Analog_Out: Frequency_to_Analog_Out;
	RAMP_WORD: RAMP_INT;
END_VAR
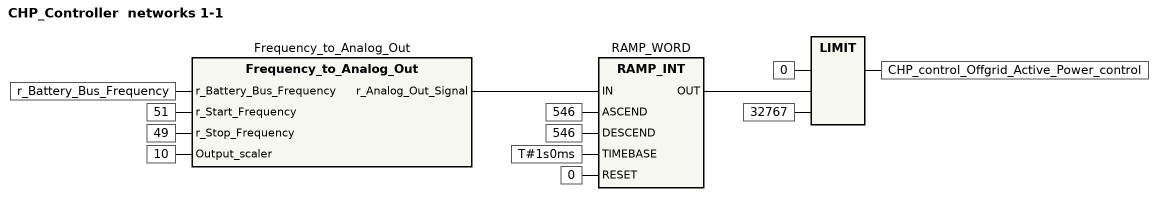
_FBD_ (* Function Block Diagram *)
NETWORK 1
	LIMIT(0, RAMP_WORD:RAMP_INT(IN: Frequency_to_Analog_Out:Frequency_to_Analog_Out(r_Battery_Bus_Frequency: r_Battery_Bus_Frequency, r_Start_Frequency: 51, r_Stop_Frequency: 49, Output_scaler: 10), ASCEND: 546, DESCEND: 546, TIMEBASE: T#1s0ms, RESET: 0), 32767) => CHP_control_Offgrid_Active_Power_control
_END_FBD_
(* the same logic as Structured Text *)
(* Network 1 *)
Frequency_to_Analog_Out(r_Battery_Bus_Frequency := r_Battery_Bus_Frequency, r_Start_Frequency := 51, r_Stop_Frequency := 49, Output_scaler := 10);
RAMP_WORD(IN := Frequency_to_Analog_Out.r_Analog_Out_Signal, ASCEND := 546, DESCEND := 546, TIMEBASE := T#1s0ms, RESET := 0);
CHP_control_Offgrid_Active_Power_control := LIMIT(0, RAMP_WORD.OUT, 32767);
END_PROGRAM

(* POU 02. Batterybus Frequency to Analog Out/Frequency_to_Analog_Out, ST *)
FUNCTION_BLOCK Frequency_to_Analog_Out
VAR_INPUT
	r_Battery_Bus_Frequency						:	REAL;
	r_Start_Frequency								:	REAL:=49;
	r_Stop_Frequency								:	REAL:=51;
	Output_scaler										:	REAL:=1;
END_VAR

VAR_OUTPUT
	r_Analog_Out_Signal								:	WORD;
END_VAR

VAR

END_VAR
(* limit control range inbetween start/stop input*)
IF r_Start_Frequency < r_Stop_Frequency THEN
	IF r_Battery_Bus_Frequency < r_Start_Frequency THEN
			r_Battery_Bus_Frequency := r_Start_Frequency;
	END_IF
	IF r_Battery_Bus_Frequency > r_Stop_Frequency THEN
			r_Battery_Bus_Frequency := r_Stop_Frequency;
	END_IF
ELSE
	IF r_Battery_Bus_Frequency > r_Start_Frequency THEN
			r_Battery_Bus_Frequency := r_Start_Frequency;
	END_IF
	IF r_Battery_Bus_Frequency < r_Stop_Frequency THEN
			r_Battery_Bus_Frequency := r_Stop_Frequency;
	END_IF
END_IF

(*r_Analog_Out_Signal := (r_Battery_Bus_Frequency - r_Start_Frequency) / (r_Stop_Frequency - r_Start_Frequency) * Output_scaler;*)
r_Analog_Out_Signal :=REAL_TO_WORD(3276.7*(r_Battery_Bus_Frequency - r_Start_Frequency) / (r_Stop_Frequency - r_Start_Frequency) * Output_scaler);
END_FUNCTION_BLOCK

(* POU SOC_to_Voltage_Out, ST *)
PROGRAM SOC_to_Voltage_Out
VAR
	Use_simulated_SOC: BOOL;
END_VAR
Use_simulated_SOC := REAL_TO_BOOL(arSystemState[310]) ;
(*TheBattery_SOC_real := 63;*)
IF Use_simulated_SOC = TRUE THEN
	other_control_control_signal := REAL_TO_WORD(3276.7*TheBattery_SOC_simulated/10);
	(*other_control_control_signal := TheBattery_SOC_simulated/10;*)
ELSE
	other_control_control_signal := REAL_TO_WORD(3276.7*TheBattery_SOC_real/10);
	(*other_control_control_signal := TheBattery_SOC_real/10;*)
END_IF
END_PROGRAM

(* POU 02. Batterybus Frequency to Analog Out/Mixer_Controller1, FBD *)
PROGRAM Mixer_Controller1
VAR
	RAMP_REAL: RAMP_REAL;
	Frequency_to_Analog_Out: Frequency_to_Analog_Out;
	RAMP_WORD2: RAMP_INT;
END_VAR
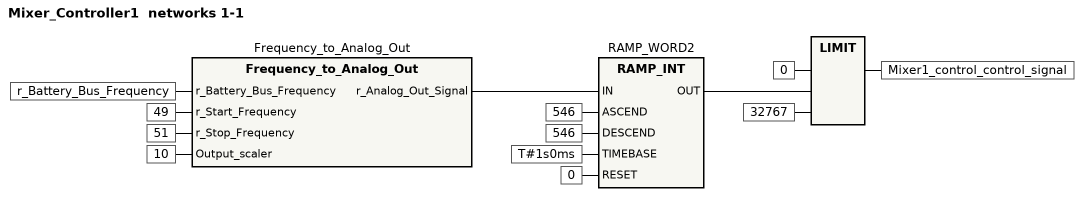
_FBD_ (* Function Block Diagram *)
NETWORK 1
	LIMIT(0, RAMP_WORD2:RAMP_INT(IN: Frequency_to_Analog_Out:Frequency_to_Analog_Out(r_Battery_Bus_Frequency: r_Battery_Bus_Frequency, r_Start_Frequency: 49, r_Stop_Frequency: 51, Output_scaler: 10), ASCEND: 546, DESCEND: 546, TIMEBASE: T#1s0ms, RESET: 0), 32767) => Mixer1_control_control_signal
_END_FBD_
(* the same logic as Structured Text *)
(* Network 1 *)
Frequency_to_Analog_Out(r_Battery_Bus_Frequency := r_Battery_Bus_Frequency, r_Start_Frequency := 49, r_Stop_Frequency := 51, Output_scaler := 10);
RAMP_WORD2(IN := Frequency_to_Analog_Out.r_Analog_Out_Signal, ASCEND := 546, DESCEND := 546, TIMEBASE := T#1s0ms, RESET := 0);
Mixer1_control_control_signal := LIMIT(0, RAMP_WORD2.OUT, 32767);
END_PROGRAM

(* POU 02. Batterybus Frequency to Analog Out/Mixer_Controller2, FBD *)
PROGRAM Mixer_Controller2
VAR
	RAMP_REAL: RAMP_REAL;
	Frequency_to_Analog_Out: Frequency_to_Analog_Out;
	RAMP_WORD3: RAMP_INT;
END_VAR
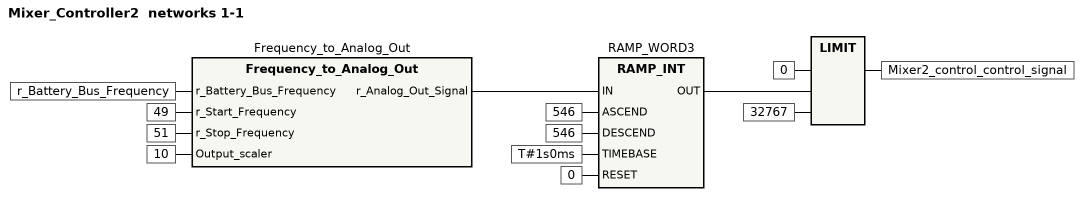
_FBD_ (* Function Block Diagram *)
NETWORK 1
	LIMIT(0, RAMP_WORD3:RAMP_INT(IN: Frequency_to_Analog_Out:Frequency_to_Analog_Out(r_Battery_Bus_Frequency: r_Battery_Bus_Frequency, r_Start_Frequency: 49, r_Stop_Frequency: 51, Output_scaler: 10), ASCEND: 546, DESCEND: 546, TIMEBASE: T#1s0ms, RESET: 0), 32767) => Mixer2_control_control_signal
_END_FBD_
(* the same logic as Structured Text *)
(* Network 1 *)
Frequency_to_Analog_Out(r_Battery_Bus_Frequency := r_Battery_Bus_Frequency, r_Start_Frequency := 49, r_Stop_Frequency := 51, Output_scaler := 10);
RAMP_WORD3(IN := Frequency_to_Analog_Out.r_Analog_Out_Signal, ASCEND := 546, DESCEND := 546, TIMEBASE := T#1s0ms, RESET := 0);
Mixer2_control_control_signal := LIMIT(0, RAMP_WORD3.OUT, 32767);
END_PROGRAM

(* POU 03. Synchroniser Switch control/run_synchroniser_swtich, ST *)
PROGRAM run_synchroniser_swtich
VAR
END_VAR
IF PQ_A.xRotatingField = PQ_B.xRotatingField THEN (* check field ration before forewarding close request *)
	SynchroniserSwitch();
END_IF

IF PQ_B.arVoltage_L_N[1] < 10 THEN (* forewarding close request when the Battery (test) bus has low voltage *)
	IF PQ_B.arVoltage_L_N[2] < 10 THEN (* forewarding close request when the Battery (test) bus has low voltage *)
		IF PQ_B.arVoltage_L_N[3] < 10 THEN (* forewarding close request when the Battery (test) bus has low voltage *)
			SynchroniserSwitch();
		END_IF
	END_IF;
END_IF
END_PROGRAM

(* POU 03. Synchroniser Switch control/SynchroniserSwitch, LD *)
PROGRAM SynchroniserSwitch
VAR
END_VAR
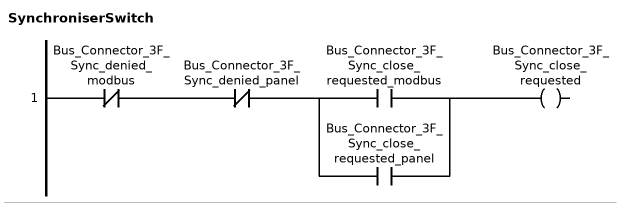
_LD_ (* Ladder Diagram *)
NETWORK 1
	[/Bus_Connector_3F_Sync_denied_modbus] - [/Bus_Connector_3F_Sync_denied_panel] - { [Bus_Connector_3F_Sync_close_requested_modbus] | [Bus_Connector_3F_Sync_close_requested_panel] } --- (Bus_Connector_3F_Sync_close_requested)
_END_LD_
(* the same logic as Structured Text *)
(* Network 1 *)
Bus_Connector_3F_Sync_close_requested := NOT Bus_Connector_3F_Sync_denied_modbus AND NOT Bus_Connector_3F_Sync_denied_panel AND (Bus_Connector_3F_Sync_close_requested_modbus OR Bus_Connector_3F_Sync_close_requested_panel);
END_PROGRAM

(* POU PLC_PRG, FBD *)
PROGRAM PLC_PRG
(*
  Function: 	Reading a CSV file
  Description: 	This project shows a functionblock which reads data from a CSV file into an array.
				Each line in the CSV contains a description and a real value.
				Each parameter  is terminated by CR LF.

---- Example CSV File -----

A_Value;245345
B_Value;0							
C_Value;8.3							
D_Value;-123439.3 						
E_Value;1						*)

VAR
	xLoad					: 	BOOL; (* Initiate load operation *)
	xSave					: 	BOOL; (* Initiate save operation *)
	sLoadStatus			: 	STRING; (* Feedback on load *)
	sSaveStatus			: 	STRING; (* Feedback on save *)
	ConfigData			: 	ARRAY [1..iMaxParams] OF  typCSV; (* Structure with the config data being loaded or saved *)
	sFileName			: 	STRING := 'config.csv'; (* Working Filename *)
	bSeperator 			: 	BYTE := 59; (* Semicolon (;) is the seperator between parameter and value. *)
	iError					: 	INT; (* Error Code for Save *)
	xWriteToSD			: 	BOOL := TRUE; (* User selectable location for file operation, on = 750-880 SD, off = internal flash *)
	sFilePath				: 	STRING; (* SD card is S:\, Internal Path is blank, but this points to the PLC folder *)
	sFilePath_Name		: 	STRING; (* Complete path + filename *)

	xReadFirstCycle		:	BOOL := TRUE;

	SetIPConfig				:	configToolFB;
	SetIP						:	configToolFB;
	SetSubnet					:	configToolFB;
	SetGateway				:	configToolFB;
	SetNTP					:	configToolFB;
	SetNTPEnable			:	configToolFB;
	SetSNMPName			:	configToolFB;
	SetSNMPDescription		:	configToolFB;
	SetSNMPLocation			:	configToolFB;
	SetSNMPContact			:	configToolFB;

	GetIPConfig				:	configToolFB;
	GetIP						:	configToolFB;
	GetSubnet					:	configToolFB;
	GetGateway				:	configToolFB;
	GetNTP					:	configToolFB;
	GetSNMPName			:	configToolFB;
	GetSNMPDescription		:	configToolFB;
	GetSNMPLocation		:	configToolFB;
	GetSNMPContact			:	configToolFB;
	GetFirmware				:	configToolFB;
	GetMACAddress			:	configToolFB;
	GetProjectDate			:	configToolFB;
	GetProjectDescription	:	configToolFB;
	GetProjectVersion			:	configToolFB;

	stSetIPConfigCallstring				:	STRING(80);
	stSetIPCallstring						:	STRING(80);
	stSetSubnetCallstring				:	STRING(80);
	stSetGatewayCallstring				:	STRING(80);
	stSetNTPCallstring					:	STRING(80);

	iSetIPConfigCallstringResult			:	INT;
	iSetIPCallstringResult				:	INT;
	iSetSubnetCallstringResult			:	INT;
	iSetGatewayCallstringResult			:	INT;
	iSetNTPCallstringResult				: 	INT;
	iSetNTPEnabledCallstringResult	:	INT;

	iGetIPConfigCallstringResult			:	INT;
	iGetIPCallstringResult				:	INT;
	iGetSubnetCallstringResult			:	INT;
	iGetGatewayCallstringResult			:	INT;
	iGetNTPCallstringResult				: 	INT;
	iGetNTPEnabledCallstringResult	:	INT;

	iGetFirmwareCallstringResult				:	INT;
	iGetMACAddressCallstringResult			:	INT;
	iGetProjectDateCallstringResult				:	INT;
	iGetProjectDescriptionCallstringResult		:	INT;
	iGetProjectVersionCallstringResult			:	INT;

	stGetIPConfigCallstring				:	STRING(80);
	stGetIPCallstring						:	STRING(80);
	stGetSubnetCallstring				:	STRING(80);
	stGetGatewayCallstring				:	STRING(80);
	stGetNTPCallstring					:	STRING(80);

	stSetIPConfigResult					:	STRING(80);
	stSetIPResult							:	STRING(80);
	stSetSubnetResult					:	STRING(80);
	stSetGatewayResult					:	STRING(80);
	stSetNTPResult						:	STRING(80);

	stGetIPConfigResult					:	STRING(80);
	stGetIPResult							:	STRING(80);
	stGetSubnetResult					:	STRING(80);
	stGetGatewayResult					:	STRING(80);
	stGetNTPResult						:	STRING(80);

	stSetSNMPNameDeviceCallstring					:	STRING(80);
	stSetSNMPDescriptionCallstring						:	STRING(80);
	stSetSNMPPhysicalLocationCallstring				:	STRING(80);
	stSetSNMPContactCallstring							:	STRING(80);

	stGetSNMPNameDeviceResult						:	STRING(80);
	stGetSNMPDescriptionResult						:	STRING(80);
	stGetSNMPPhysicalLocationResult					:	STRING(80);
	stGetSNMPContactResult							:	STRING(80);

	stGetFirmwareResult									:	STRING(80);
	stGetMACAddressResult								:	STRING(80);
	stGetProjectDateResult								:	STRING(80);
	stGetProjectDescriptionResult						:	STRING(80);
	stGetProjectVersionResult							:	STRING(80);

	iSetSNMPNameDeviceCallstringResult				:	INT;
	iSetSNMPDescriptionCallstringResult				:	INT;
	iSetSNMPPhysicalLocationCallstringResult			:	INT;
	iSetSNMPContactCallstringResult					:	INT;

	iGetSNMPNameDeviceCallstringResult				:	INT;
	iGetSNMPDescriptionCallstringResult				:	INT;
	iGetSNMPPhysicalLocationCallstringResult			:	INT;
	iGetSNMPContactCallstringResult					:	INT;

	CurrentTimeDate										:	STRING;

END_VAR
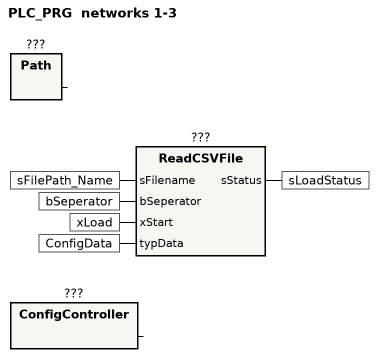
_FBD_ (* Function Block Diagram *)
NETWORK 1
	???:Path()
NETWORK 2
	???:ReadCSVFile(sFilename: sFilePath_Name, bSeperator: bSeperator, xStart: xLoad, typData: ConfigData) => sLoadStatus
NETWORK 3
	???:ConfigController()
_END_FBD_
END_PROGRAM
ACTION ConfigController:
IF xReadFirstCycle = TRUE THEN

	(*xLoad := TRUE;*)

	IF sLoadStatus = 'Data read OK' THEN
	
		(* Set Ethernet settings of controller *)
		
		(* Set static IP-Address*)
		
		
			SetIPConfig(
			bEnable:= TRUE,
			stCallString:= 'config_interfaces interface=X1 config-type=static state=enabled',
			stResultString=> stSetIPConfigResult,
			iFbResult=> iSetIPCallstringResult );
		
		(* Set IP-Address of controller *)
		
			stSetIPCallstring := CONCAT('config_interfaces interface X1 ip-address=',stIPAddressEthernet);
		
			SetIP(
			bEnable:= TRUE,
			stCallString:= stSetIPCallstring ,
			stResultString=> stSetIPResult,
			iFbResult=> iSetIPCallstringResult );
		
		(* Set Subnet-Address of controller *)
		
			stSetSubnetCallstring := CONCAT('config_interfaces interface X1 subnet-mask=',stIPAddressSubnet);
		
			SetSubnet(
			bEnable:= TRUE,
			stCallString:= stSetSubnetCallstring ,
			iFbResult=> iSetSubnetCallstringResult );
		
		(* Set Gateway-Address of controller *)
		
			stSetGatewayCallstring := CONCAT('config_default_gateway interface=X1 default-gateway-value=', stIPAddressGateway);
		
			SetGateway(
			bEnable:= TRUE,
			stCallString:= stSetGatewayCallstring ,
			iFbResult=> iSetGatewayCallstringResult );
		
		(* Set NTP-Address of controller *)
		
			SetNTPEnable(
			bEnable:= TRUE,
			stCallString:= 'config_sntp state=enabled' ,
			iFbResult=> iSetNTPEnabledCallstringResult );
		
			stSetNTPCallstring := CONCAT('config_sntp time-server=',stIPAddressNTP);
		
			SetNTP(
			bEnable:= TRUE,
			stCallString:= stSetNTPCallstring ,
			iFbResult=> iSetNTPCallstringResult );
		
		(* Set SNMP-configuration of the controller *)
		
		(* Set SNMP-description of the controller *)
		
			stSetSNMPDescriptionCallstring := CONCAT('config_snmp description=',stSNMPDescription);
		
			SetSNMPDescription(
			bEnable:= TRUE,
			stCallString:= stSetSNMPDescriptionCallstring,
			iFbResult=> iSetSNMPDescriptionCallstringResult );
		
		(* Set SNMP-name of the controller *)
		
			stSetSNMPNameDeviceCallstring := CONCAT('config_snmp device-name=',stSNMPNameDevice);
		
			SetSNMPName(
			bEnable:= TRUE,
			stCallString:= stSetSNMPNameDeviceCallstring,
			iFbResult=> iSetSNMPNameDeviceCallstringResult );
		
		(* Set SNMP-location of the controller *)

			stSetSNMPPhysicalLocationCallstring := CONCAT('config_snmp physical-location=',stSNMPPhysicalLocation);
		
			SetSNMPLocation(
			bEnable:= TRUE,
			stCallString:= stSetSNMPPhysicalLocationCallstring,
			iFbResult=> iSetSNMPPhysicalLocationCallstringResult);
		
		(* Set SNMP-contact information of the controller *)
		
			stSetSNMPContactCallstring := CONCAT('config_snmp contact=',stSNMPcontact);
		
			SetSNMPContact(
			bEnable:= TRUE,
			stCallString:= stSetSNMPContactCallstring,
			iFbResult=> iSetSNMPContactCallstringResult);
		
			xReadFirstCycle := FALSE;
			xLoad := FALSE;

	END_IF

END_IF

(* Get Ethernet settings of controller *)

(* Get IP-configuration of controller *)

	GetIPConfig(
	bEnable:= TRUE,
	stCallString:= 'get_eth_config X1 config-type' ,
	stResultString=> stGetIPConfigResult,
	iFbResult=> iGetIPConfigCallstringResult );

(* Get IP-Address of controller *)

	GetIP(
	bEnable:= TRUE,
	stCallString:= 'get_eth_config X1 ip-address' ,
	stResultString=> stGetIPResult,
	iFbResult=> iGetIPCallstringResult );

(* Get Subnet-Address of controller *)

	GetSubnet(
	bEnable:= TRUE,
	stCallString:= 'get_eth_config X1 subnet-mask' ,
	stResultString=> stGetSubnetResult,
	iFbResult=> iGetSubnetCallstringResult );

(* Get Gateway-Address of controller *)

	GetGateway(
	bEnable:= TRUE,
	stCallString:= 'get_eth_config X1 default-gateway' ,
	stResultString=> stGetGatewayResult,
	iFbResult=> iGetGatewayCallstringResult );

(* Get NTP-Address of controller *)

	GetNTP(
	bEnable:= TRUE,
	stCallString:= 'get_ntp_config time-server' ,
	stResultString=> stGetNTPResult,
	iFbResult=> iGetNTPCallstringResult );

(* Get SNMP-configuration of the controller *)

(* Get SNMP-description of the controller *)

	GetSNMPDescription(
	bEnable:= TRUE,
	stCallString:= 'get_snmp_data description',
	stResultString=> stGetSNMPDescriptionResult,
	iFbResult=> iGetSNMPDescriptionCallstringResult );

(* Get SNMP-description of the controller *)

	GetSNMPName(
	bEnable:= TRUE,
	stCallString:= 'get_snmp_data device-name',
	stResultString=> stGetSNMPNameDeviceResult,
	iFbResult=> iGetSNMPNameDeviceCallstringResult );

(* Get SNMP-location of the controller *)

	GetSNMPLocation(
	bEnable:= TRUE,
	stCallString:= 'get_snmp_data physical-location',
	stResultString=> stGetSNMPPhysicalLocationResult,
	iFbResult=> iGetSNMPPhysicalLocationCallstringResult);

(* Get SNMP-contact information of the controller *)

	GetSNMPContact(
	bEnable:= TRUE,
	stCallString:= 'get_snmp_data contact',
	stResultString=> stGetSNMPContactResult,
	iFbResult=> iGetSNMPContactCallstringResult);

(* Get Firmware information of the controller *)

	GetFirmware(
	bEnable:= TRUE,
	stCallString:= 'get_coupler_details firmware-revision',
	stResultString=> stGetFirmwareResult,
	iFbResult=> iGetFirmwareCallstringResult);

(* Get MAC-Address of the controller *)

	GetMACAddress(
	bEnable:= TRUE,
	stCallString:= 'get_actual_eth_config X1 mac-address',
	stResultString=> stGetMACAddressResult,
	iFbResult=> iGetMACAddressCallstringResult);

(* Get Project Date of the controller *)

	GetProjectDate(
	bEnable:= TRUE,
	stCallString:= 'get_rts_info project date',
	stResultString=> stGetProjectDateResult,
	iFbResult=> iGetProjectDateCallstringResult);

(* Get Project Description of the controller *)

	GetProjectDescription(
	bEnable:= TRUE,
	stCallString:= 'get_rts_info project description',
	stResultString=> stGetProjectDescriptionResult,
	iFbResult=> iGetProjectDescriptionCallstringResult);

(* Get Project version of the controller *)

	GetProjectVersion(
	bEnable:= TRUE,
	stCallString:= 'get_rts_info project version',
	stResultString=> stGetProjectVersionResult,
	iFbResult=> iGetProjectVersionCallstringResult);

	CurrentTimeDate := Date_Time();
END_ACTION
ACTION Path:
IF xWriteToSD THEN
	sFilePath := '/media/sd/';
ELSE
	sFilePath := '';
END_IF
sFilePath_Name := CONCAT(sFilePath, sFileName);
END_ACTION
ACTION SetParam:
	stIPAddressEthernet := ConfigData[1].Parameter[1];
	stIPAddressSubnet  := ConfigData[2].Parameter[1];
	stIPAddressGateway  := ConfigData[3].Parameter[1];
	stIPAddressNTP := ConfigData[4].Parameter[1];

	stSNMPNameDevice := ConfigData[5].Parameter[1];
	stSNMPDescription := ConfigData[6].Parameter[1];
	stSNMPPhysicalLocation := ConfigData[7].Parameter[1];
	stSNMPContact := ConfigData[8].Parameter[1];
END_ACTION

(* POU 08. SD CARD logging/ReadCSVFile, ST *)
PROGRAM ReadCSVFile
VAR_INPUT
	sFilename		:STRING;
	bSeperator		:BYTE:=59;(*seperator semicolon:59=;*)
END_VAR
VAR_IN_OUT
	xStart			:BOOL;
	typData			:ARRAY [1..iMaxParams] OF  typCSV;
END_VAR
VAR_OUTPUT
	sStatus			:STRING;
END_VAR
VAR
	bEndOfFile		:BYTE:=13;
	FileIdent		:DWORD;
	rawdata			:ARRAY[0..gc_RawDataSize] OF BYTE;
	filesizev		:DINT;
	tempstring		:STRING;
	startposition	:INT;
	i				:INT;
	j				:INT;
	k				:INT;
END_VAR
IF xStart THEN
	FileIdent:=SysFileOpen(FileName:=sFilename, Mode:='r');
	IF fileident<>0 THEN
		SysFileRead(File:=Fileident, Buffer:=ADR(rawdata), Size:=SIZEOF(rawdata));
		filesizev:=SysFileGetSize(FileName:=sFilename);
		IF filesizev>gc_RawDataSize THEN
			filesizev:=gc_RawDataSize;
		END_IF
		SysFileClose(File:=fileident);(*this function is blocking*)
	ELSE
		sStatus:='File does not exist';
		xStart:=FALSE;
		RETURN;(*no such file available*)
	END_IF
(*copy data to typData array*)
	startposition:=0;
	i:=0;
	FOR j:=1 TO iMaxParams DO
		(*First value in dataset is of type DT. The following value is seperated by bSeperator*)
		WHILE rawdata[startposition+i]<>bSeperator DO
			i:=i+1;
		END_WHILE
		rawdata[startposition+i]:=0;
		MEMCPY(pSourceAddress:=ADR(rawdata[startposition]), pDestinationAddress:=ADR(tempstring), BytesToCopy:=i+1);
		typdata[j].sDescription:=tempstring;
		startposition:=startposition+i+1;
		i:=0;
		(*The parameter values are of type word. The following values are seperated by bSeperator*)
		FOR k:=1 TO gc_ParameterCount-1 DO
			WHILE rawdata[startposition+i]<>bSeperator DO
				i:=i+1;
			END_WHILE
			rawdata[startposition+i]:=0;
			MEMCPY(pSourceAddress:=ADR(rawdata[startposition]), pDestinationAddress:=ADR(tempstring), BytesToCopy:=i+1);
			typdata[j].Parameter[k]:=(tempstring);
			startposition:=startposition+i+1;
			i:=0;
		END_FOR
		(*Copying the last parameter from typ word. The data set is terminated by CR LF*)
		WHILE rawdata[startposition+i]<>bEndOfFile DO
			i:=i+1;
		END_WHILE
		rawdata[startposition+i]:=0;
		MEMCPY(pSourceAddress:=ADR(rawdata[startposition]), pDestinationAddress:=ADR(tempstring), BytesToCopy:=i+1);
		typdata[j].Parameter[k]:=(tempstring);
		startposition:=startposition+i+2;(*The data set is terminated by CR LF(13,10)*)
		i:=0;
	END_FOR
(*copy data to typData array finished*)
	sStatus:='Data read OK';
	xStart:=FALSE;
END_IF
END_PROGRAM

(* POU 02. Batterybus Frequency to Analog Out/EV_Controller, FBD *)
PROGRAM EV_Controller
VAR
	RAMP_REAL: RAMP_REAL;
	Frequency_to_Analog_Out: Frequency_to_Analog_Out;
	EV_control_control_signal2: INT;
	RAMP_WORD4: RAMP_INT;
END_VAR
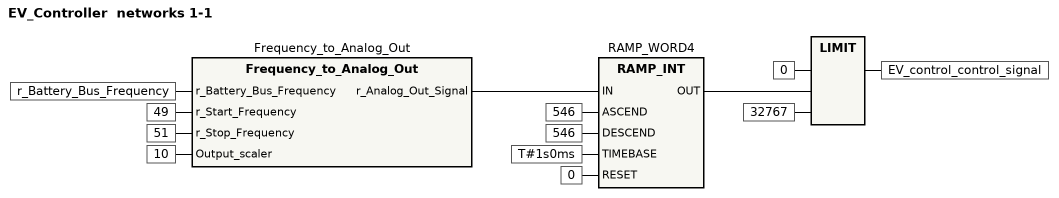
_FBD_ (* Function Block Diagram *)
NETWORK 1
	LIMIT(0, RAMP_WORD4:RAMP_INT(IN: Frequency_to_Analog_Out:Frequency_to_Analog_Out(r_Battery_Bus_Frequency: r_Battery_Bus_Frequency, r_Start_Frequency: 49, r_Stop_Frequency: 51, Output_scaler: 10), ASCEND: 546, DESCEND: 546, TIMEBASE: T#1s0ms, RESET: 0), 32767) => EV_control_control_signal
_END_FBD_
(* the same logic as Structured Text *)
(* Network 1 *)
Frequency_to_Analog_Out(r_Battery_Bus_Frequency := r_Battery_Bus_Frequency, r_Start_Frequency := 49, r_Stop_Frequency := 51, Output_scaler := 10);
RAMP_WORD4(IN := Frequency_to_Analog_Out.r_Analog_Out_Signal, ASCEND := 546, DESCEND := 546, TIMEBASE := T#1s0ms, RESET := 0);
EV_control_control_signal := LIMIT(0, RAMP_WORD4.OUT, 32767);
END_PROGRAM

(* POU Configuration/MODBUS_CONFIGURATION, ST *)
PROGRAM MODBUS_CONFIGURATION
VAR                                
END_VAR                            
(*                                 
   <?xml version="1.0" encoding="UTF-16" standalone="yes"?>
<network xml_structure_version="1" xml_feature_version="1">
	<generator_settings minRTUTaskCycleTimeMs="100" minEthaskCycleTimeMs="5" ethSlaveMultiplier="0.1" rtuInterfaceMultiplier="0.1" taskGeneration="false"/>
	<master_interface type="eth" name="" expanded="true">
		<mb_slave comment="" name="Janitza_UMG5090" expanded="true" type="generic">
			<mb_connection type="eth" transport="UDP" port="502" ip="192.168.1.2" unitid="1" request_delay_ms="0" response_timeout_ms="20"/>
			<generic_vars comment="" expanded="true">
				<generic_var data_type="REAL">
					<generic_params name="PactiveL1" comment="" expanded="false" mb_iotype="unused" mb_access="ro" var_byteorder="B3B4B1B2"/>
					<mb_address explicitAccess="false" FCRead="3" FCWrite="0" ReadMBAddress="2069" WriteMBAddress="0" ReadBitOffset="0" WriteBitOffset="0"/>
				</generic_var>
				<generic_var data_type="REAL">
					<generic_params name="PactiveL2" comment="" expanded="true" mb_iotype="unused" mb_access="ro" var_byteorder="B3B4B1B2"/>
					<mb_address explicitAccess="false" FCRead="3" FCWrite="0" ReadMBAddress="2071" WriteMBAddress="0" ReadBitOffset="0" WriteBitOffset="0"/>
				</generic_var>
				<generic_var data_type="REAL">
					<generic_params name="PactiveL3" comment="" expanded="true" mb_iotype="unused" mb_access="ro" var_byteorder="B3B4B1B2"/>
					<mb_address explicitAccess="false" FCRead="3" FCWrite="0" ReadMBAddress="2073" WriteMBAddress="0" ReadBitOffset="0" WriteBitOffset="0"/>
				</generic_var>
				<generic_var data_type="REAL">
					<generic_params name="PreactiveL1" comment="" expanded="false" mb_iotype="unused" mb_access="ro" var_byteorder="B3B4B1B2"/>
					<mb_address explicitAccess="false" FCRead="3" FCWrite="0" ReadMBAddress="2077" WriteMBAddress="0" ReadBitOffset="0" WriteBitOffset="0"/>
				</generic_var>
				<generic_var data_type="REAL">
					<generic_params name="PreactiveL2" comment="" expanded="true" mb_iotype="unused" mb_access="ro" var_byteorder="B3B4B1B2"/>
					<mb_address explicitAccess="false" FCRead="3" FCWrite="0" ReadMBAddress="2079" WriteMBAddress="0" ReadBitOffset="0" WriteBitOffset="0"/>
				</generic_var>
				<generic_var data_type="REAL">
					<generic_params name="PreactiveL3" comment="" expanded="true" mb_iotype="unused" mb_access="ro" var_byteorder="B3B4B1B2"/>
					<mb_address explicitAccess="false" FCRead="3" FCWrite="0" ReadMBAddress="2081" WriteMBAddress="0" ReadBitOffset="0" WriteBitOffset="0"/>
				</generic_var>
				<generic_var data_type="REAL">
					<generic_params name="VoltageL1" comment="" expanded="true" mb_iotype="unused" mb_access="ro" var_byteorder="B3B4B1B2"/>
					<mb_address explicitAccess="false" FCRead="3" FCWrite="0" ReadMBAddress="2053" WriteMBAddress="0" ReadBitOffset="0" WriteBitOffset="0"/>
				</generic_var>
				<generic_var data_type="REAL">
					<generic_params name="VoltageL2" comment="" expanded="false" mb_iotype="unused" mb_access="ro" var_byteorder="B3B4B1B2"/>
					<mb_address explicitAccess="false" FCRead="3" FCWrite="0" ReadMBAddress="2055" WriteMBAddress="0" ReadBitOffset="0" WriteBitOffset="0"/>
				</generic_var>
				<generic_var data_type="REAL">
					<generic_params name="VoltageL3" comment="" expanded="false" mb_iotype="unused" mb_access="ro" var_byteorder="B3B4B1B2"/>
					<mb_address explicitAccess="false" FCRead="3" FCWrite="0" ReadMBAddress="2057" WriteMBAddress="0" ReadBitOffset="0" WriteBitOffset="0"/>
				</generic_var>
				<generic_var data_type="REAL">
					<generic_params name="VoltageL4" comment="" expanded="false" mb_iotype="unused" mb_access="ro" var_byteorder="B3B4B1B2"/>
					<mb_address explicitAccess="false" FCRead="3" FCWrite="0" ReadMBAddress="2059" WriteMBAddress="0" ReadBitOffset="0" WriteBitOffset="0"/>
				</generic_var>
				<generic_var data_type="REAL">
					<generic_params name="PhaseCurrentL1" comment="" expanded="true" mb_iotype="unused" mb_access="ro" var_byteorder="B3B4B1B2"/>
					<mb_address explicitAccess="false" FCRead="3" FCWrite="0" ReadMBAddress="2061" WriteMBAddress="0" ReadBitOffset="0" WriteBitOffset="0"/>
				</generic_var>
				<generic_var data_type="REAL">
					<generic_params name="PhaseCurrentL2" comment="" expanded="true" mb_iotype="unused" mb_access="ro" var_byteorder="B3B4B1B2"/>
					<mb_address explicitAccess="false" FCRead="3" FCWrite="0" ReadMBAddress="2063" WriteMBAddress="0" ReadBitOffset="0" WriteBitOffset="0"/>
				</generic_var>
				<generic_var data_type="REAL">
					<generic_params name="PhaseCurrentL3" comment="" expanded="true" mb_iotype="unused" mb_access="ro" var_byteorder="B3B4B1B2"/>
					<mb_address explicitAccess="false" FCRead="3" FCWrite="0" ReadMBAddress="2065" WriteMBAddress="0" ReadBitOffset="0" WriteBitOffset="0"/>
				</generic_var>
				<generic_var data_type="REAL">
					<generic_params name="PhaseCurrentLN" comment="" expanded="true" mb_iotype="unused" mb_access="ro" var_byteorder="B3B4B1B2"/>
					<mb_address explicitAccess="false" FCRead="3" FCWrite="0" ReadMBAddress="2067" WriteMBAddress="0" ReadBitOffset="0" WriteBitOffset="0"/>
				</generic_var>
				<generic_var data_type="REAL">
					<generic_params name="FieldRotation" comment="" expanded="true" mb_iotype="unused" mb_access="ro" var_byteorder="B3B4B1B2"/>
					<mb_address explicitAccess="false" FCRead="3" FCWrite="0" ReadMBAddress="2185" WriteMBAddress="0" ReadBitOffset="0" WriteBitOffset="0"/>
				</generic_var>
				<generic_var data_type="REAL">
					<generic_params name="CosPihL1" comment="" expanded="true" mb_iotype="unused" mb_access="ro" var_byteorder="B3B4B1B2"/>
					<mb_address explicitAccess="false" FCRead="3" FCWrite="0" ReadMBAddress="2159" WriteMBAddress="0" ReadBitOffset="0" WriteBitOffset="0"/>
				</generic_var>
				<generic_var data_type="REAL">
					<generic_params name="CosPihL2" comment="" expanded="true" mb_iotype="unused" mb_access="ro" var_byteorder="B3B4B1B2"/>
					<mb_address explicitAccess="false" FCRead="3" FCWrite="0" ReadMBAddress="2161" WriteMBAddress="0" ReadBitOffset="0" WriteBitOffset="0"/>
				</generic_var>
				<generic_var data_type="REAL">
					<generic_params name="CosPihL3" comment="" expanded="true" mb_iotype="unused" mb_access="ro" var_byteorder="B3B4B1B2"/>
					<mb_address explicitAccess="false" FCRead="3" FCWrite="0" ReadMBAddress="2163" WriteMBAddress="0" ReadBitOffset="0" WriteBitOffset="0"/>
				</generic_var>
				<generic_var data_type="REAL">
					<generic_params name="Frequency" comment="" expanded="true" mb_iotype="unused" mb_access="ro" var_byteorder="B3B4B1B2"/>
					<mb_address explicitAccess="false" FCRead="3" FCWrite="0" ReadMBAddress="2175" WriteMBAddress="0" ReadBitOffset="0" WriteBitOffset="0"/>
				</generic_var>
				<generic_var data_type="REAL">
					<generic_params name="PactivetTot" comment="" expanded="false" mb_iotype="unused" mb_access="ro" var_byteorder="B3B4B1B2"/>
					<mb_address explicitAccess="false" FCRead="3" FCWrite="0" ReadMBAddress="2105" WriteMBAddress="0" ReadBitOffset="0" WriteBitOffset="0"/>
				</generic_var>
				<generic_var data_type="REAL">
					<generic_params name="PactivetTotL4" comment="" expanded="false" mb_iotype="unused" mb_access="ro" var_byteorder="B3B4B1B2"/>
					<mb_address explicitAccess="false" FCRead="3" FCWrite="0" ReadMBAddress="2113" WriteMBAddress="0" ReadBitOffset="0" WriteBitOffset="0"/>
				</generic_var>
			</generic_vars>
		</mb_slave>
	</master_interface>
</network>
                              
*)                                 
;                                  
END_PROGRAM

(* POU 02. Batterybus Frequency to Analog Out/other_control_signal, FBD *)
PROGRAM other_control_signal
VAR
	RAMP_REAL: RAMP_REAL;
	Frequency_to_Analog_Out: Frequency_to_Analog_Out;
END_VAR
